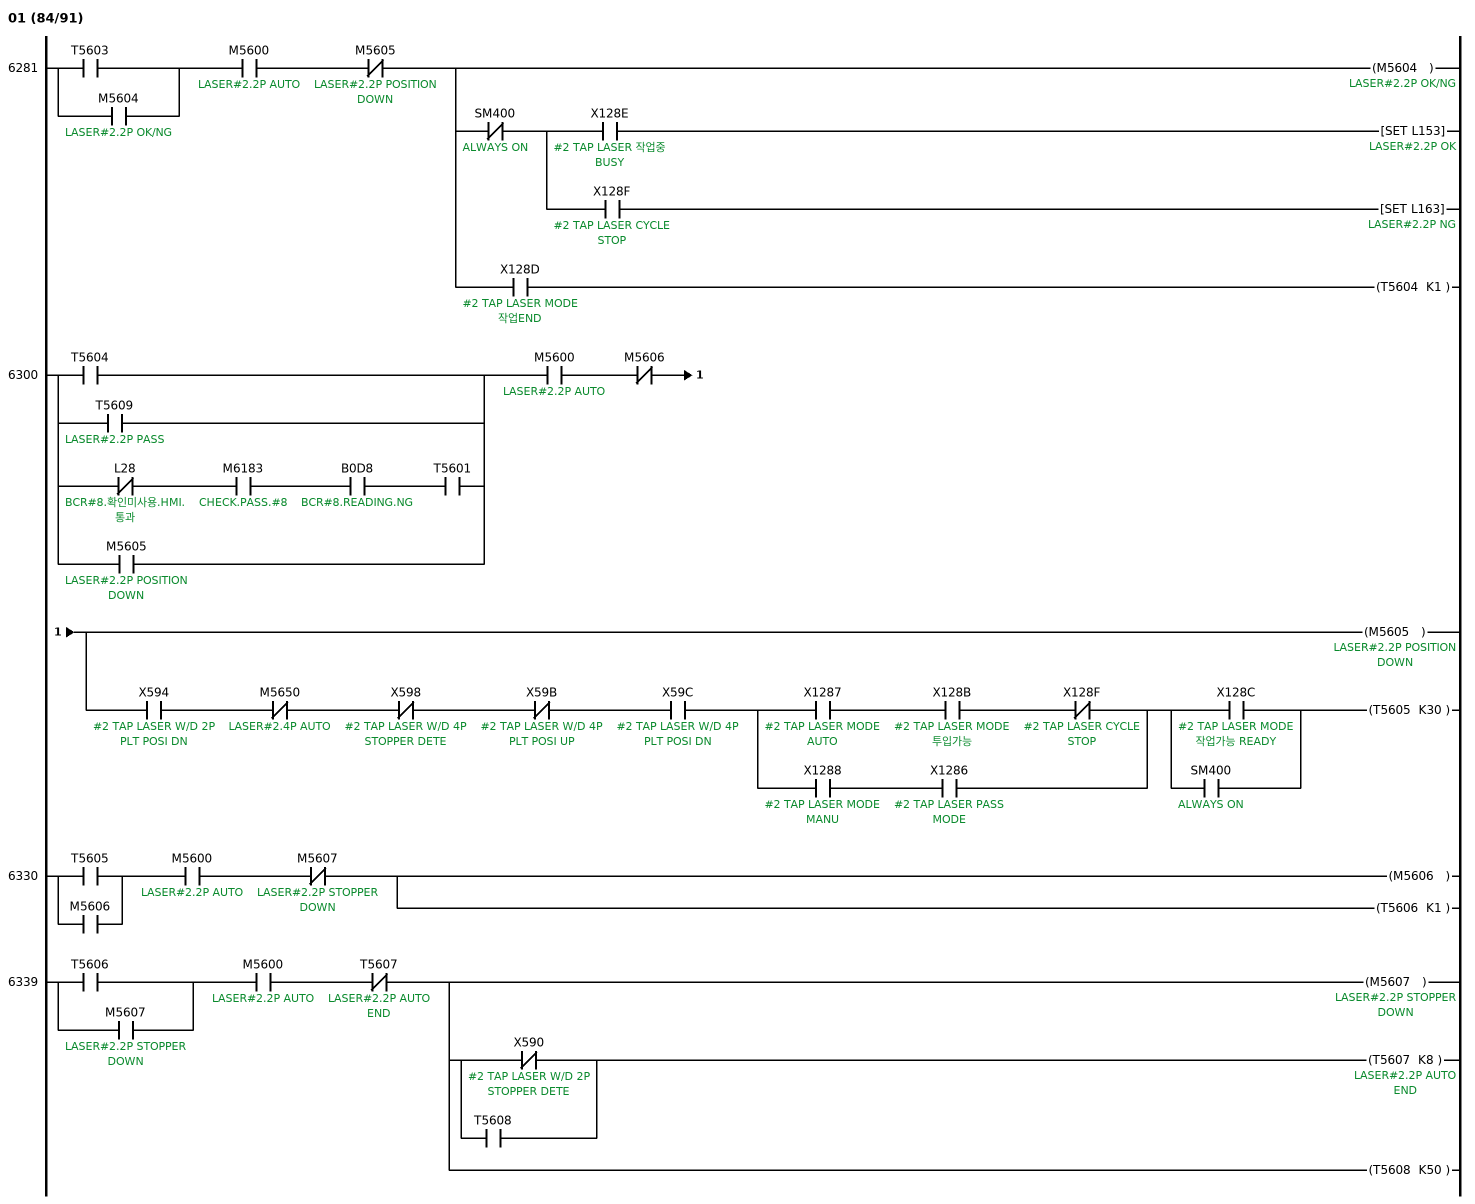
6281  LD      T5603
      OR      M5604  ; LASER#2.2P OK/NG
      AND     M5600  ; LASER#2.2P AUTO
      ANI     M5605  ; LASER#2.2P POSITION DOWN
      OUT     M5604  ; LASER#2.2P OK/NG
      MPS
      ANI     SM400  ; ALWAYS ON
      MPS
      AND     X128E  ; #2 TAP LASER 작업중 BUSY
      SET     L153  ; LASER#2.2P OK
      MPP
      AND     X128F  ; #2 TAP LASER CYCLE STOP
      SET     L163  ; LASER#2.2P NG
      MPP
      AND     X128D  ; #2 TAP LASER MODE 작업END
      OUT     T5604 K1
6300  LD      T5604
      OR      T5609  ; LASER#2.2P PASS
      LDI     L28  ; BCR#8.확인미사용.HMI.통과
      AND     M6183  ; CHECK.PASS.#8
      AND     B0D8  ; BCR#8.READING.NG
      AND     T5601
      ORB
      OR      M5605  ; LASER#2.2P POSITION DOWN
      AND     M5600  ; LASER#2.2P AUTO
      ANI     M5606
      OUT     M5605  ; LASER#2.2P POSITION DOWN
      AND     X594  ; #2 TAP LASER W/D 2P PLT POSI DN
      ANI     M5650  ; LASER#2.4P AUTO
      ANI     X598  ; #2 TAP LASER W/D 4P STOPPER DETE
      ANI     X59B  ; #2 TAP LASER W/D 4P PLT POSI UP
      AND     X59C  ; #2 TAP LASER W/D 4P PLT POSI DN
      LD      X1287  ; #2 TAP LASER MODE AUTO
      AND     X128B  ; #2 TAP LASER MODE 투입가능
      ANI     X128F  ; #2 TAP LASER CYCLE STOP
      LD      X1288  ; #2 TAP LASER MODE MANU
      AND     X1286  ; #2 TAP LASER PASS MODE
      ORB
      ANB
      LD      X128C  ; #2 TAP LASER MODE 작업가능 READY
      OR      SM400  ; ALWAYS ON
      ANB
      OUT     T5605 K30
6330  LD      T5605
      OR      M5606
      AND     M5600  ; LASER#2.2P AUTO
      ANI     M5607  ; LASER#2.2P STOPPER DOWN
      OUT     M5606
      OUT     T5606 K1
6339  LD      T5606
      OR      M5607  ; LASER#2.2P STOPPER DOWN
      AND     M5600  ; LASER#2.2P AUTO
      ANI     T5607  ; LASER#2.2P AUTO END
      OUT     M5607  ; LASER#2.2P STOPPER DOWN
      MPS
      LDI     X590  ; #2 TAP LASER W/D 2P STOPPER DETE
      OR      T5608
      ANB
      OUT     T5607 K8  ; LASER#2.2P AUTO END
      MPP
      OUT     T5608 K50
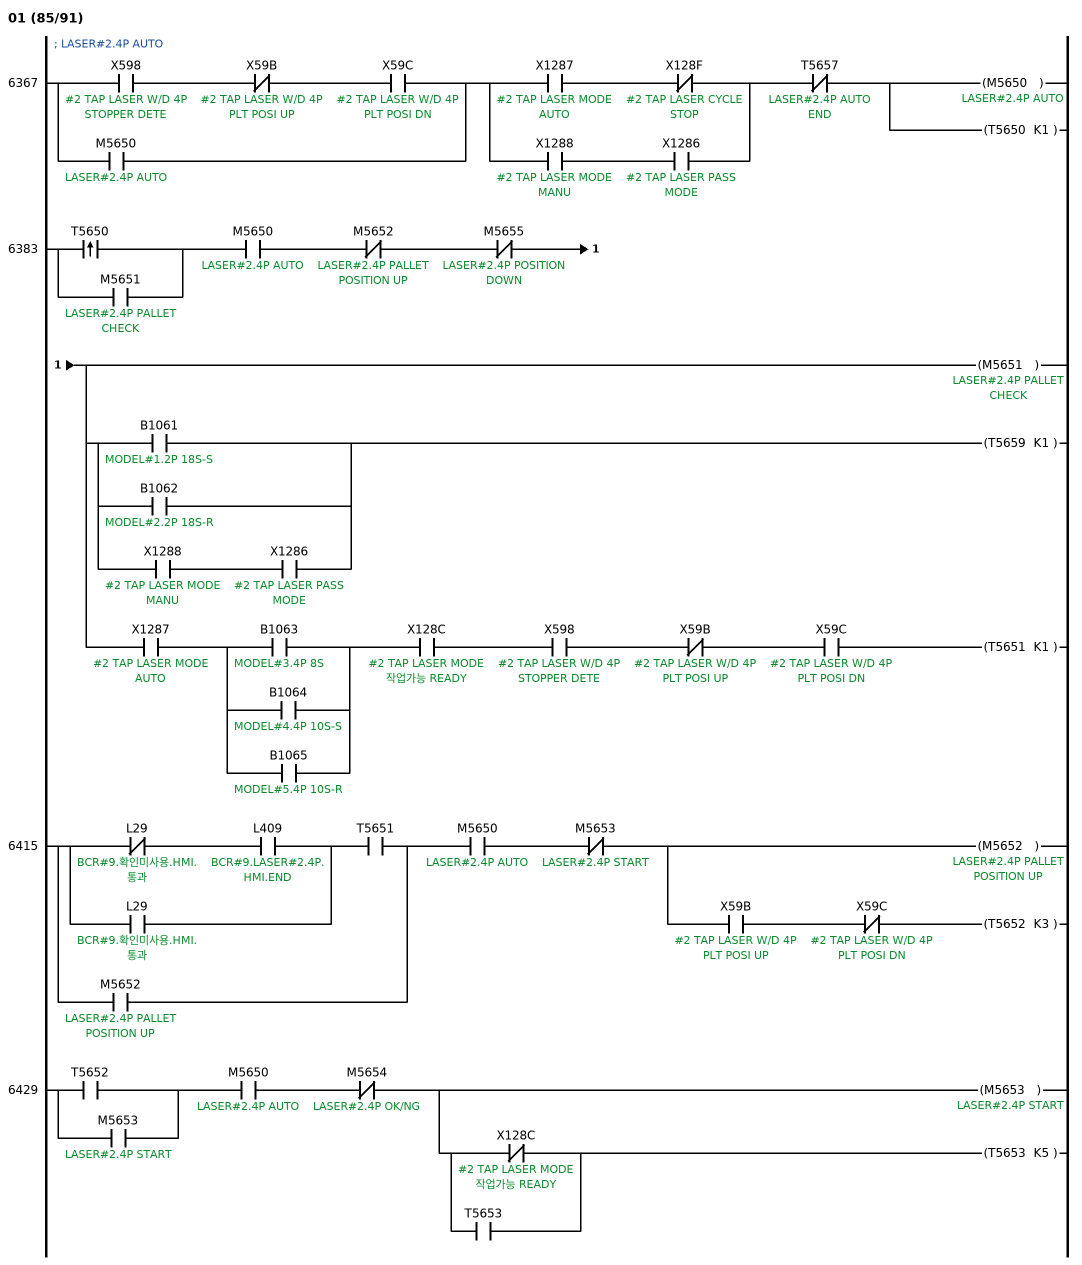
; LASER#2.4P AUTO
6367  LD      X598  ; #2 TAP LASER W/D 4P STOPPER DETE
      ANI     X59B  ; #2 TAP LASER W/D 4P PLT POSI UP
      AND     X59C  ; #2 TAP LASER W/D 4P PLT POSI DN
      OR      M5650  ; LASER#2.4P AUTO
      LD      X1287  ; #2 TAP LASER MODE AUTO
      ANI     X128F  ; #2 TAP LASER CYCLE STOP
      LD      X1288  ; #2 TAP LASER MODE MANU
      AND     X1286  ; #2 TAP LASER PASS MODE
      ORB
      ANB
      ANI     T5657  ; LASER#2.4P AUTO END
      OUT     M5650  ; LASER#2.4P AUTO
      OUT     T5650 K1
6383  LDP     T5650
      OR      M5651  ; LASER#2.4P PALLET CHECK
      AND     M5650  ; LASER#2.4P AUTO
      ANI     M5652  ; LASER#2.4P PALLET POSITION UP
      ANI     M5655  ; LASER#2.4P POSITION DOWN
      OUT     M5651  ; LASER#2.4P PALLET CHECK
      MPS
      LD      B1061  ; MODEL#1.2P 18S-S
      OR      B1062  ; MODEL#2.2P 18S-R
      LD      X1288  ; #2 TAP LASER MODE MANU
      AND     X1286  ; #2 TAP LASER PASS MODE
      ORB
      ANB
      OUT     T5659 K1
      MPP
      AND     X1287  ; #2 TAP LASER MODE AUTO
      LD      B1063  ; MODEL#3.4P 8S
      OR      B1064  ; MODEL#4.4P 10S-S
      OR      B1065  ; MODEL#5.4P 10S-R
      ANB
      AND     X128C  ; #2 TAP LASER MODE 작업가능 READY
      AND     X598  ; #2 TAP LASER W/D 4P STOPPER DETE
      ANI     X59B  ; #2 TAP LASER W/D 4P PLT POSI UP
      AND     X59C  ; #2 TAP LASER W/D 4P PLT POSI DN
      OUT     T5651 K1
6415  LDI     L29  ; BCR#9.확인미사용.HMI.통과
      AND     L409  ; BCR#9.LASER#2.4P.HMI.END
      OR      L29  ; BCR#9.확인미사용.HMI.통과
      AND     T5651
      OR      M5652  ; LASER#2.4P PALLET POSITION UP
      AND     M5650  ; LASER#2.4P AUTO
      ANI     M5653  ; LASER#2.4P START
      OUT     M5652  ; LASER#2.4P PALLET POSITION UP
      AND     X59B  ; #2 TAP LASER W/D 4P PLT POSI UP
      ANI     X59C  ; #2 TAP LASER W/D 4P PLT POSI DN
      OUT     T5652 K3
6429  LD      T5652
      OR      M5653  ; LASER#2.4P START
      AND     M5650  ; LASER#2.4P AUTO
      ANI     M5654  ; LASER#2.4P OK/NG
      OUT     M5653  ; LASER#2.4P START
      LDI     X128C  ; #2 TAP LASER MODE 작업가능 READY
      OR      T5653
      ANB
      OUT     T5653 K5
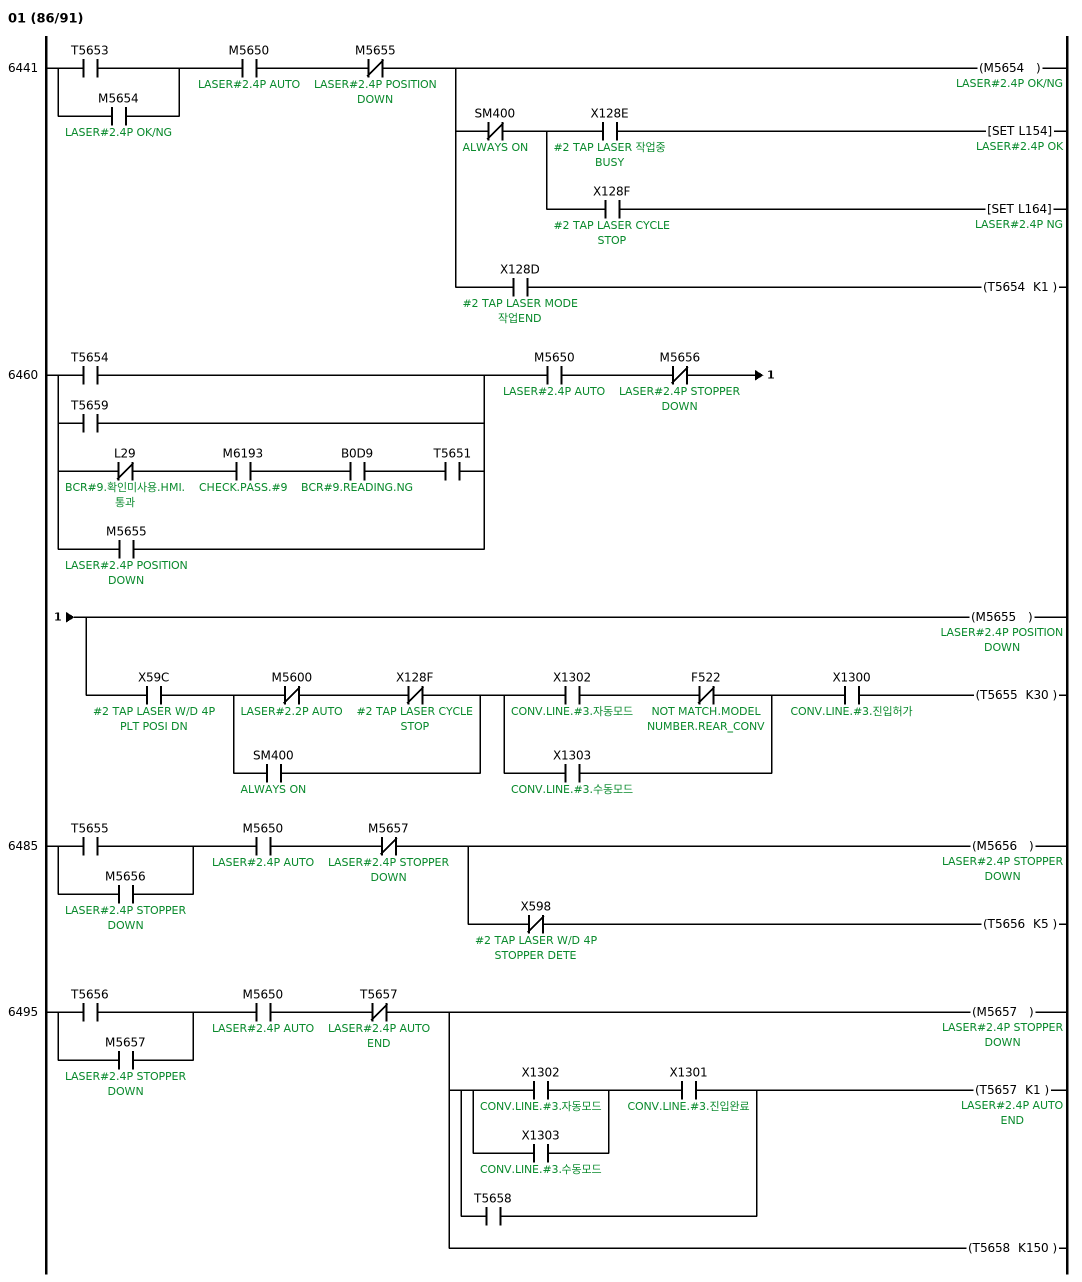
6441  LD      T5653
      OR      M5654  ; LASER#2.4P OK/NG
      AND     M5650  ; LASER#2.4P AUTO
      ANI     M5655  ; LASER#2.4P POSITION DOWN
      OUT     M5654  ; LASER#2.4P OK/NG
      MPS
      ANI     SM400  ; ALWAYS ON
      MPS
      AND     X128E  ; #2 TAP LASER 작업중 BUSY
      SET     L154  ; LASER#2.4P OK
      MPP
      AND     X128F  ; #2 TAP LASER CYCLE STOP
      SET     L164  ; LASER#2.4P NG
      MPP
      AND     X128D  ; #2 TAP LASER MODE 작업END
      OUT     T5654 K1
6460  LD      T5654
      OR      T5659
      LDI     L29  ; BCR#9.확인미사용.HMI.통과
      AND     M6193  ; CHECK.PASS.#9
      AND     B0D9  ; BCR#9.READING.NG
      AND     T5651
      ORB
      OR      M5655  ; LASER#2.4P POSITION DOWN
      AND     M5650  ; LASER#2.4P AUTO
      ANI     M5656  ; LASER#2.4P STOPPER DOWN
      OUT     M5655  ; LASER#2.4P POSITION DOWN
      AND     X59C  ; #2 TAP LASER W/D 4P PLT POSI DN
      LDI     M5600  ; LASER#2.2P AUTO
      ANI     X128F  ; #2 TAP LASER CYCLE STOP
      OR      SM400  ; ALWAYS ON
      ANB
      LD      X1302  ; CONV.LINE.#3.자동모드
      ANI     F522  ; NOT MATCH.MODEL NUMBER.REAR_CONV
      OR      X1303  ; CONV.LINE.#3.수동모드
      ANB
      AND     X1300  ; CONV.LINE.#3.진입허가
      OUT     T5655 K30
6485  LD      T5655
      OR      M5656  ; LASER#2.4P STOPPER DOWN
      AND     M5650  ; LASER#2.4P AUTO
      ANI     M5657  ; LASER#2.4P STOPPER DOWN
      OUT     M5656  ; LASER#2.4P STOPPER DOWN
      ANI     X598  ; #2 TAP LASER W/D 4P STOPPER DETE
      OUT     T5656 K5
6495  LD      T5656
      OR      M5657  ; LASER#2.4P STOPPER DOWN
      AND     M5650  ; LASER#2.4P AUTO
      ANI     T5657  ; LASER#2.4P AUTO END
      OUT     M5657  ; LASER#2.4P STOPPER DOWN
      MPS
      LD      X1302  ; CONV.LINE.#3.자동모드
      OR      X1303  ; CONV.LINE.#3.수동모드
      AND     X1301  ; CONV.LINE.#3.진입완료
      OR      T5658
      ANB
      OUT     T5657 K1  ; LASER#2.4P AUTO END
      MPP
      OUT     T5658 K150
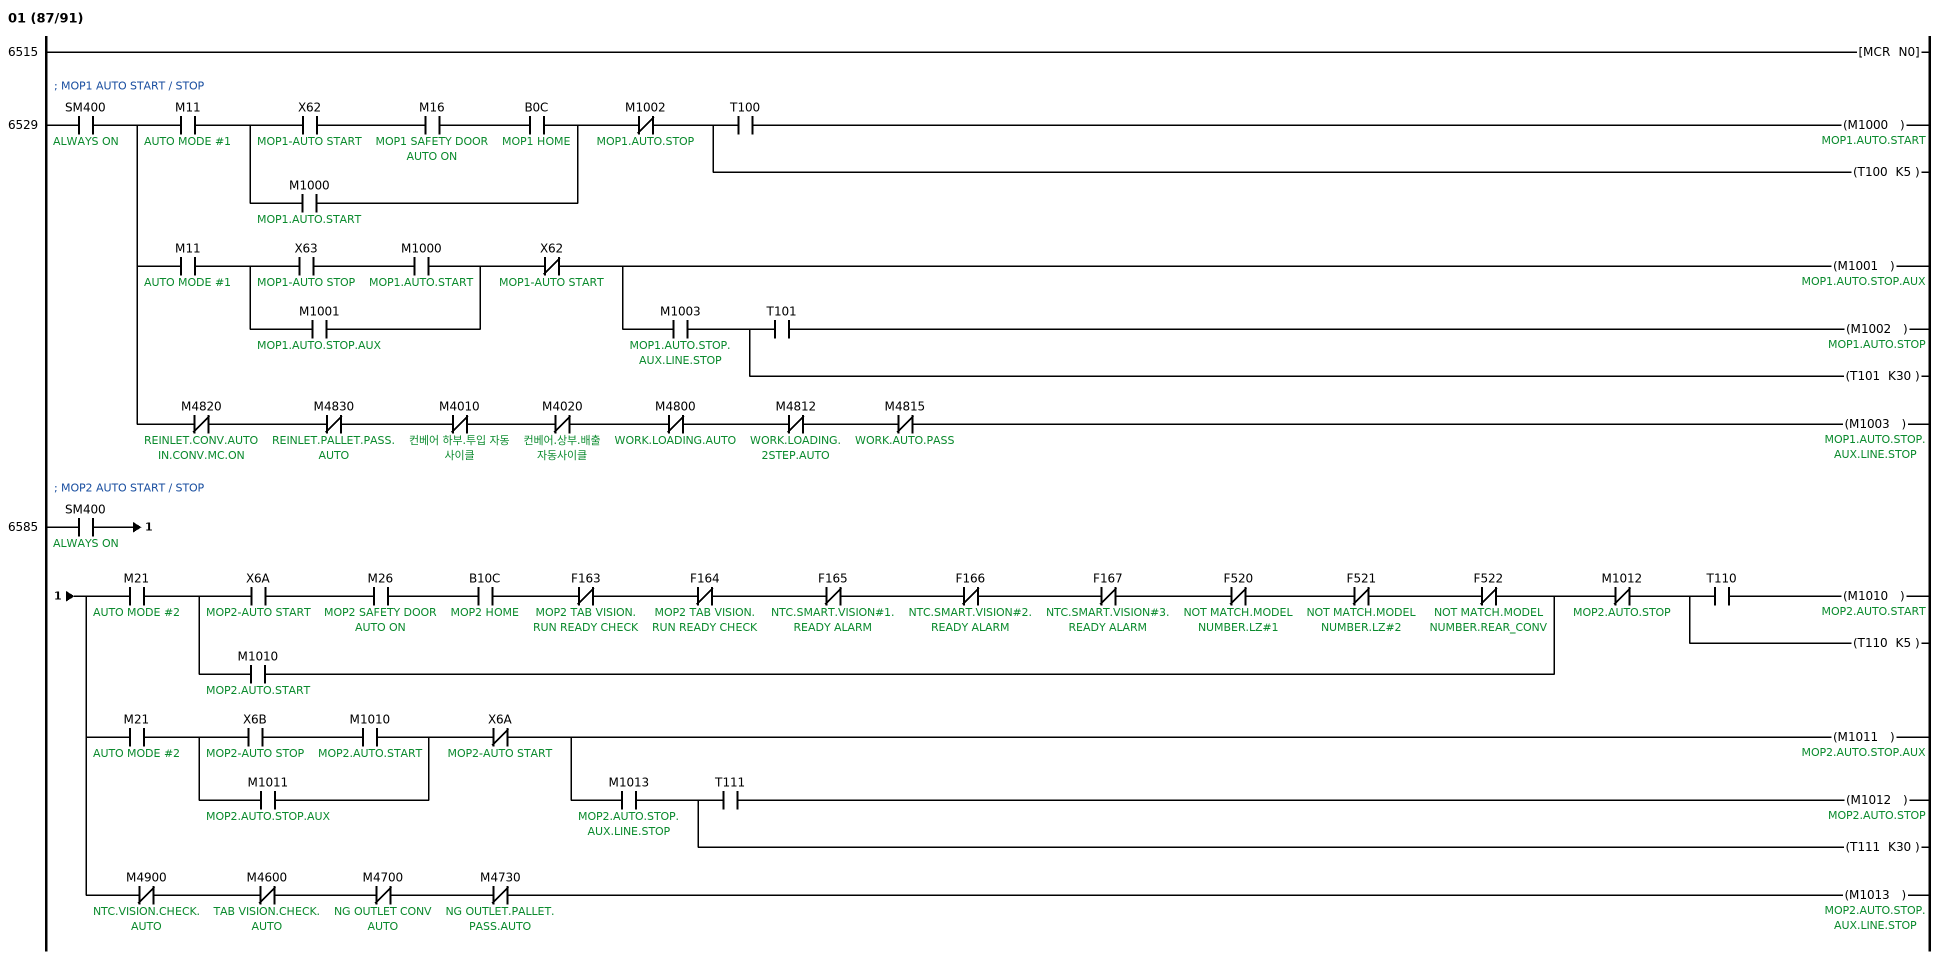
6515  MCR     N0
; MOP1 AUTO START / STOP
6529  LD      SM400  ; ALWAYS ON
      MPS
      AND     M11  ; AUTO MODE #1
      LD      X62  ; MOP1-AUTO START
      AND     M16  ; MOP1 SAFETY DOOR AUTO ON
      AND     B0C  ; MOP1 HOME
      OR      M1000  ; MOP1.AUTO.START
      ANB
      ANI     M1002  ; MOP1.AUTO.STOP
      MPS
      AND     T100
      OUT     M1000  ; MOP1.AUTO.START
      MPP
      OUT     T100 K5
      MRD
      AND     M11  ; AUTO MODE #1
      LD      X63  ; MOP1-AUTO STOP
      AND     M1000  ; MOP1.AUTO.START
      OR      M1001  ; MOP1.AUTO.STOP.AUX
      ANB
      ANI     X62  ; MOP1-AUTO START
      OUT     M1001  ; MOP1.AUTO.STOP.AUX
      AND     M1003  ; MOP1.AUTO.STOP.AUX.LINE.STOP
      MPS
      AND     T101
      OUT     M1002  ; MOP1.AUTO.STOP
      MPP
      OUT     T101 K30
      MPP
      ANI     M4820  ; REINLET.CONV.AUTO IN.CONV.MC.ON
      ANI     M4830  ; REINLET.PALLET.PASS.AUTO
      ANI     M4010  ; 컨베어 하부.투입 자동 사이클
      ANI     M4020  ; 컨베어.상부.배출 자동사이클
      ANI     M4800  ; WORK.LOADING.AUTO
      ANI     M4812  ; WORK.LOADING.2STEP.AUTO
      ANI     M4815  ; WORK.AUTO.PASS
      OUT     M1003  ; MOP1.AUTO.STOP.AUX.LINE.STOP
; MOP2 AUTO START / STOP
6585  LD      SM400  ; ALWAYS ON
      MPS
      AND     M21  ; AUTO MODE #2
      LD      X6A  ; MOP2-AUTO START
      AND     M26  ; MOP2 SAFETY DOOR AUTO ON
      AND     B10C  ; MOP2 HOME
      ANI     F163  ; MOP2 TAB VISION. RUN READY CHECK
      ANI     F164  ; MOP2 TAB VISION. RUN READY CHECK
      ANI     F165  ; NTC.SMART.VISION#1.READY ALARM
      ANI     F166  ; NTC.SMART.VISION#2.READY ALARM
      ANI     F167  ; NTC.SMART.VISION#3.READY ALARM
      ANI     F520  ; NOT MATCH.MODEL NUMBER.LZ#1
      ANI     F521  ; NOT MATCH.MODEL NUMBER.LZ#2
      ANI     F522  ; NOT MATCH.MODEL NUMBER.REAR_CONV
      OR      M1010  ; MOP2.AUTO.START
      ANB
      ANI     M1012  ; MOP2.AUTO.STOP
      MPS
      AND     T110
      OUT     M1010  ; MOP2.AUTO.START
      MPP
      OUT     T110 K5
      MRD
      AND     M21  ; AUTO MODE #2
      LD      X6B  ; MOP2-AUTO STOP
      AND     M1010  ; MOP2.AUTO.START
      OR      M1011  ; MOP2.AUTO.STOP.AUX
      ANB
      ANI     X6A  ; MOP2-AUTO START
      OUT     M1011  ; MOP2.AUTO.STOP.AUX
      AND     M1013  ; MOP2.AUTO.STOP.AUX.LINE.STOP
      MPS
      AND     T111
      OUT     M1012  ; MOP2.AUTO.STOP
      MPP
      OUT     T111 K30
      MPP
      ANI     M4900  ; NTC.VISION.CHECK.AUTO
      ANI     M4600  ; TAB VISION.CHECK.AUTO
      ANI     M4700  ; NG OUTLET CONV AUTO
      ANI     M4730  ; NG OUTLET.PALLET.PASS.AUTO
      OUT     M1013  ; MOP2.AUTO.STOP.AUX.LINE.STOP
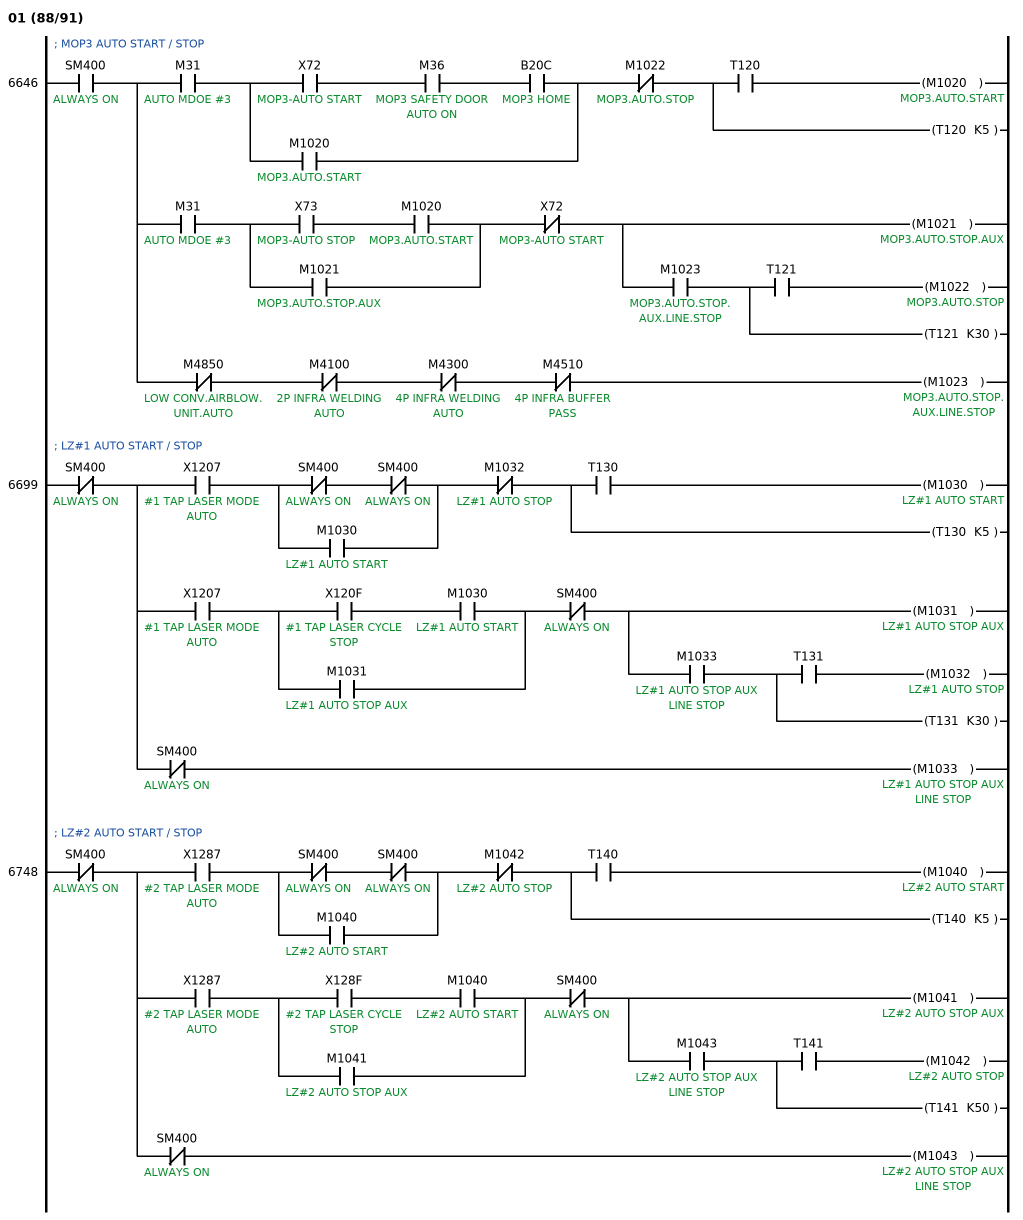
; MOP3 AUTO START / STOP
6646  LD      SM400  ; ALWAYS ON
      MPS
      AND     M31  ; AUTO MDOE #3
      LD      X72  ; MOP3-AUTO START
      AND     M36  ; MOP3 SAFETY DOOR AUTO ON
      AND     B20C  ; MOP3 HOME
      OR      M1020  ; MOP3.AUTO.START
      ANB
      ANI     M1022  ; MOP3.AUTO.STOP
      MPS
      AND     T120
      OUT     M1020  ; MOP3.AUTO.START
      MPP
      OUT     T120 K5
      MRD
      AND     M31  ; AUTO MDOE #3
      LD      X73  ; MOP3-AUTO STOP
      AND     M1020  ; MOP3.AUTO.START
      OR      M1021  ; MOP3.AUTO.STOP.AUX
      ANB
      ANI     X72  ; MOP3-AUTO START
      OUT     M1021  ; MOP3.AUTO.STOP.AUX
      AND     M1023  ; MOP3.AUTO.STOP.AUX.LINE.STOP
      MPS
      AND     T121
      OUT     M1022  ; MOP3.AUTO.STOP
      MPP
      OUT     T121 K30
      MPP
      ANI     M4850  ; LOW CONV.AIRBLOW.UNIT.AUTO
      ANI     M4100  ; 2P INFRA WELDING AUTO
      ANI     M4300  ; 4P INFRA WELDING AUTO
      ANI     M4510  ; 4P INFRA BUFFER PASS
      OUT     M1023  ; MOP3.AUTO.STOP.AUX.LINE.STOP
; LZ#1 AUTO START / STOP
6699  LDI     SM400  ; ALWAYS ON
      MPS
      AND     X1207  ; #1 TAP LASER MODE AUTO
      LDI     SM400  ; ALWAYS ON
      ANI     SM400  ; ALWAYS ON
      OR      M1030  ; LZ#1 AUTO START
      ANB
      ANI     M1032  ; LZ#1 AUTO STOP
      MPS
      AND     T130
      OUT     M1030  ; LZ#1 AUTO START
      MPP
      OUT     T130 K5
      MRD
      AND     X1207  ; #1 TAP LASER MODE AUTO
      LD      X120F  ; #1 TAP LASER CYCLE STOP
      AND     M1030  ; LZ#1 AUTO START
      OR      M1031  ; LZ#1 AUTO STOP AUX
      ANB
      ANI     SM400  ; ALWAYS ON
      OUT     M1031  ; LZ#1 AUTO STOP AUX
      AND     M1033  ; LZ#1 AUTO STOP AUX LINE STOP
      MPS
      AND     T131
      OUT     M1032  ; LZ#1 AUTO STOP
      MPP
      OUT     T131 K30
      MPP
      ANI     SM400  ; ALWAYS ON
      OUT     M1033  ; LZ#1 AUTO STOP AUX LINE STOP
; LZ#2 AUTO START / STOP
6748  LDI     SM400  ; ALWAYS ON
      MPS
      AND     X1287  ; #2 TAP LASER MODE AUTO
      LDI     SM400  ; ALWAYS ON
      ANI     SM400  ; ALWAYS ON
      OR      M1040  ; LZ#2 AUTO START
      ANB
      ANI     M1042  ; LZ#2 AUTO STOP
      MPS
      AND     T140
      OUT     M1040  ; LZ#2 AUTO START
      MPP
      OUT     T140 K5
      MRD
      AND     X1287  ; #2 TAP LASER MODE AUTO
      LD      X128F  ; #2 TAP LASER CYCLE STOP
      AND     M1040  ; LZ#2 AUTO START
      OR      M1041  ; LZ#2 AUTO STOP AUX
      ANB
      ANI     SM400  ; ALWAYS ON
      OUT     M1041  ; LZ#2 AUTO STOP AUX
      AND     M1043  ; LZ#2 AUTO STOP AUX LINE STOP
      MPS
      AND     T141
      OUT     M1042  ; LZ#2 AUTO STOP
      MPP
      OUT     T141 K50
      MPP
      ANI     SM400  ; ALWAYS ON
      OUT     M1043  ; LZ#2 AUTO STOP AUX LINE STOP
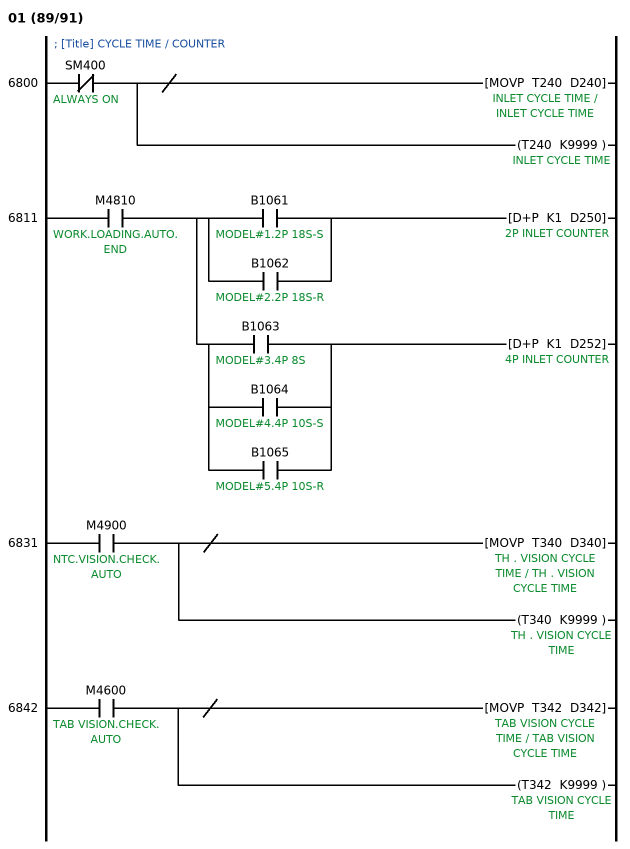
; [Title] CYCLE TIME / COUNTER
6800  LDI     SM400  ; ALWAYS ON
      MPS
      INV
      MOVP    T240 D240  ; INLET CYCLE TIME / INLET CYCLE TIME
      MPP
      OUT     T240 K9999  ; INLET CYCLE TIME
6811  LD      M4810  ; WORK.LOADING.AUTO.END
      MPS
      LD      B1061  ; MODEL#1.2P 18S-S
      OR      B1062  ; MODEL#2.2P 18S-R
      ANB
      D+P     K1 D250  ; 2P INLET COUNTER
      MPP
      LD      B1063  ; MODEL#3.4P 8S
      OR      B1064  ; MODEL#4.4P 10S-S
      OR      B1065  ; MODEL#5.4P 10S-R
      ANB
      D+P     K1 D252  ; 4P INLET COUNTER
6831  LD      M4900  ; NTC.VISION.CHECK.AUTO
      MPS
      INV
      MOVP    T340 D340  ; TH . VISION CYCLE TIME / TH . VISION CYCLE TIME
      MPP
      OUT     T340 K9999  ; TH . VISION CYCLE TIME
6842  LD      M4600  ; TAB VISION.CHECK.AUTO
      MPS
      INV
      MOVP    T342 D342  ; TAB VISION CYCLE TIME / TAB VISION CYCLE TIME
      MPP
      OUT     T342 K9999  ; TAB VISION CYCLE TIME
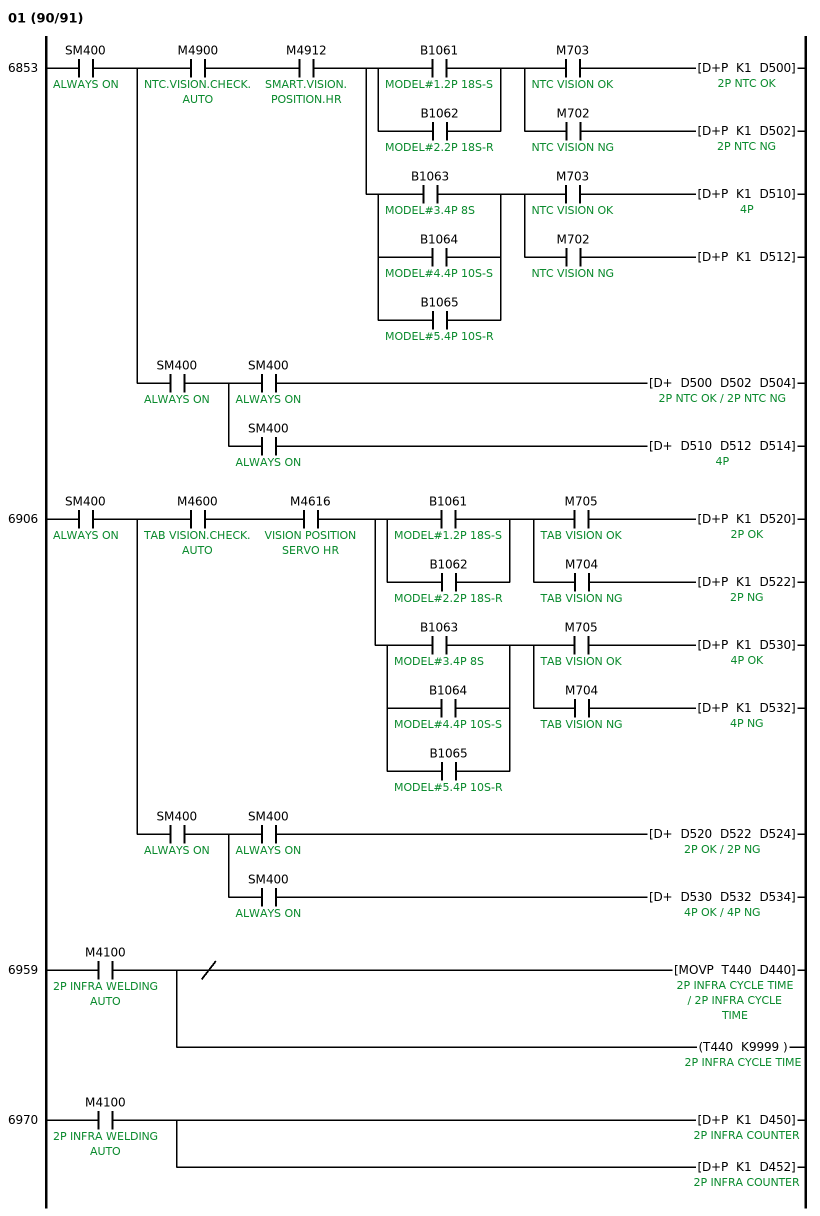
6853  LD      SM400  ; ALWAYS ON
      MPS
      AND     M4900  ; NTC.VISION.CHECK.AUTO
      AND     M4912  ; SMART.VISION.POSITION.HR
      MPS
      LD      B1061  ; MODEL#1.2P 18S-S
      OR      B1062  ; MODEL#2.2P 18S-R
      ANB
      MPS
      AND     M703  ; NTC VISION OK
      D+P     K1 D500  ; 2P NTC OK
      MPP
      AND     M702  ; NTC VISION NG
      D+P     K1 D502  ; 2P NTC NG
      MPP
      LD      B1063  ; MODEL#3.4P 8S
      OR      B1064  ; MODEL#4.4P 10S-S
      OR      B1065  ; MODEL#5.4P 10S-R
      ANB
      MPS
      AND     M703  ; NTC VISION OK
      D+P     K1 D510  ; 4P
      MPP
      AND     M702  ; NTC VISION NG
      D+P     K1 D512
      MPP
      AND     SM400  ; ALWAYS ON
      MPS
      AND     SM400  ; ALWAYS ON
      D+      D500 D502 D504
      MPP
      AND     SM400  ; ALWAYS ON
      D+      D510 D512 D514
6906  LD      SM400  ; ALWAYS ON
      MPS
      AND     M4600  ; TAB VISION.CHECK.AUTO
      AND     M4616  ; VISION POSITION SERVO HR
      MPS
      LD      B1061  ; MODEL#1.2P 18S-S
      OR      B1062  ; MODEL#2.2P 18S-R
      ANB
      MPS
      AND     M705  ; TAB VISION OK
      D+P     K1 D520  ; 2P OK
      MPP
      AND     M704  ; TAB VISION NG
      D+P     K1 D522  ; 2P NG
      MPP
      LD      B1063  ; MODEL#3.4P 8S
      OR      B1064  ; MODEL#4.4P 10S-S
      OR      B1065  ; MODEL#5.4P 10S-R
      ANB
      MPS
      AND     M705  ; TAB VISION OK
      D+P     K1 D530  ; 4P OK
      MPP
      AND     M704  ; TAB VISION NG
      D+P     K1 D532  ; 4P NG
      MPP
      AND     SM400  ; ALWAYS ON
      MPS
      AND     SM400  ; ALWAYS ON
      D+      D520 D522 D524
      MPP
      AND     SM400  ; ALWAYS ON
      D+      D530 D532 D534
6959  LD      M4100  ; 2P INFRA WELDING AUTO
      MPS
      INV
      MOVP    T440 D440  ; 2P INFRA CYCLE TIME / 2P INFRA CYCLE TIME
      MPP
      OUT     T440 K9999  ; 2P INFRA CYCLE TIME
6970  LD      M4100  ; 2P INFRA WELDING AUTO
      D+P     K1 D450  ; 2P INFRA COUNTER
      D+P     K1 D452  ; 2P INFRA COUNTER
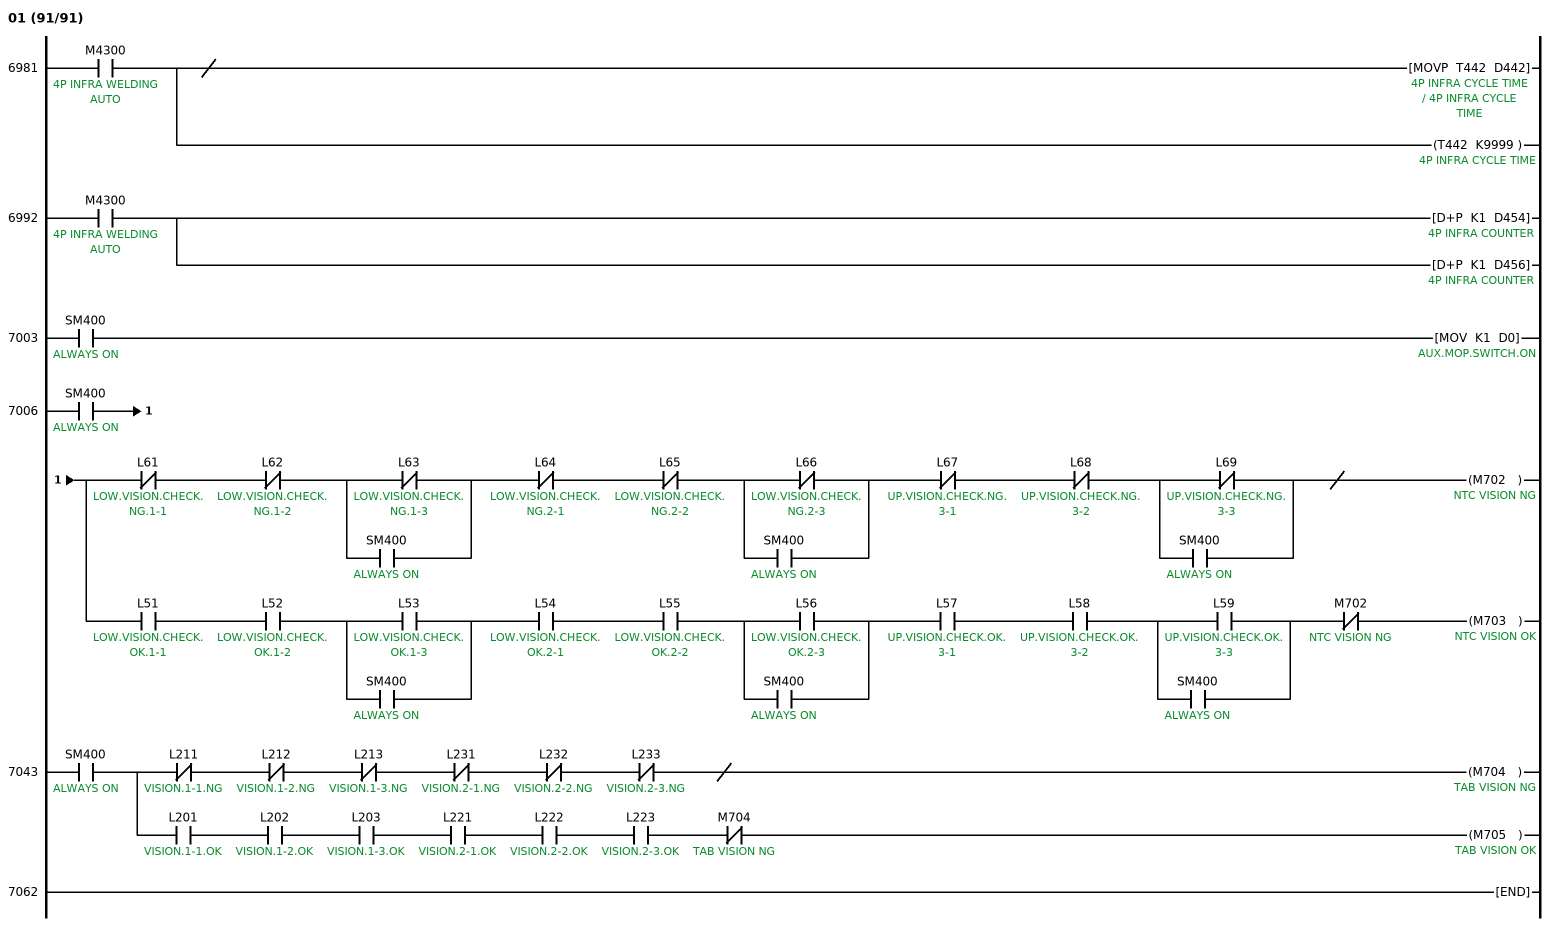
6981  LD      M4300  ; 4P INFRA WELDING AUTO
      MPS
      INV
      MOVP    T442 D442  ; 4P INFRA CYCLE TIME / 4P INFRA CYCLE TIME
      MPP
      OUT     T442 K9999  ; 4P INFRA CYCLE TIME
6992  LD      M4300  ; 4P INFRA WELDING AUTO
      D+P     K1 D454  ; 4P INFRA COUNTER
      D+P     K1 D456  ; 4P INFRA COUNTER
7003  LD      SM400  ; ALWAYS ON
      MOV     K1 D0  ; AUX.MOP.SWITCH.ON
7006  LD      SM400  ; ALWAYS ON
      MPS
      ANI     L61  ; LOW.VISION.CHECK.NG.1-1
      ANI     L62  ; LOW.VISION.CHECK.NG.1-2
      LDI     L63  ; LOW.VISION.CHECK.NG.1-3
      OR      SM400  ; ALWAYS ON
      ANB
      ANI     L64  ; LOW.VISION.CHECK.NG.2-1
      ANI     L65  ; LOW.VISION.CHECK.NG.2-2
      LDI     L66  ; LOW.VISION.CHECK.NG.2-3
      OR      SM400  ; ALWAYS ON
      ANB
      ANI     L67  ; UP.VISION.CHECK.NG.3-1
      ANI     L68  ; UP.VISION.CHECK.NG.3-2
      LDI     L69  ; UP.VISION.CHECK.NG.3-3
      OR      SM400  ; ALWAYS ON
      ANB
      INV
      OUT     M702  ; NTC VISION NG
      MPP
      AND     L51  ; LOW.VISION.CHECK.OK.1-1
      AND     L52  ; LOW.VISION.CHECK.OK.1-2
      LD      L53  ; LOW.VISION.CHECK.OK.1-3
      OR      SM400  ; ALWAYS ON
      ANB
      AND     L54  ; LOW.VISION.CHECK.OK.2-1
      AND     L55  ; LOW.VISION.CHECK.OK.2-2
      LD      L56  ; LOW.VISION.CHECK.OK.2-3
      OR      SM400  ; ALWAYS ON
      ANB
      AND     L57  ; UP.VISION.CHECK.OK.3-1
      AND     L58  ; UP.VISION.CHECK.OK.3-2
      LD      L59  ; UP.VISION.CHECK.OK.3-3
      OR      SM400  ; ALWAYS ON
      ANB
      ANI     M702  ; NTC VISION NG
      OUT     M703  ; NTC VISION OK
7043  LD      SM400  ; ALWAYS ON
      MPS
      ANI     L211  ; VISION.1-1.NG
      ANI     L212  ; VISION.1-2.NG
      ANI     L213  ; VISION.1-3.NG
      ANI     L231  ; VISION.2-1.NG
      ANI     L232  ; VISION.2-2.NG
      ANI     L233  ; VISION.2-3.NG
      INV
      OUT     M704  ; TAB VISION NG
      MPP
      AND     L201  ; VISION.1-1.OK
      AND     L202  ; VISION.1-2.OK
      AND     L203  ; VISION.1-3.OK
      AND     L221  ; VISION.2-1.OK
      AND     L222  ; VISION.2-2.OK
      AND     L223  ; VISION.2-3.OK
      ANI     M704  ; TAB VISION NG
      OUT     M705  ; TAB VISION OK
7062  END
END_PROGRAM

PROGRAM 05  // HMI
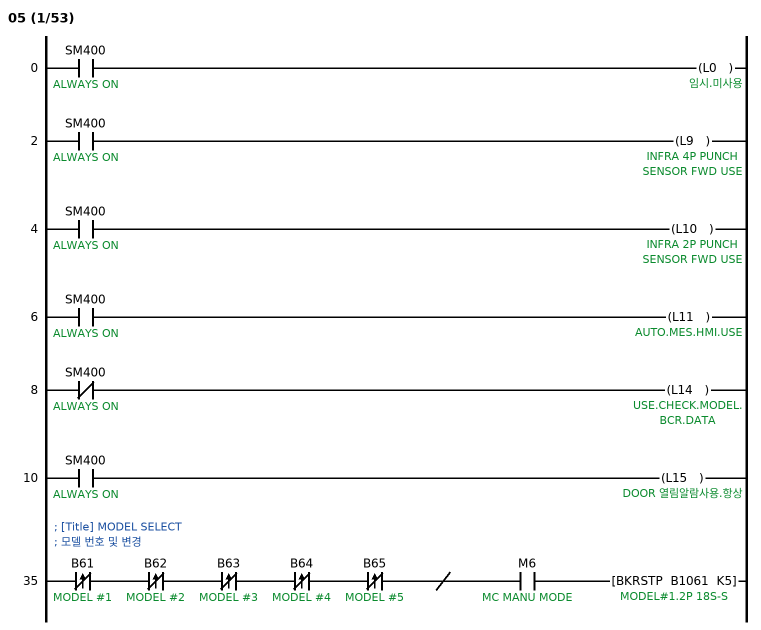
0     LD      SM400  ; ALWAYS ON
      OUT     L0  ; 임시.미사용
2     LD      SM400  ; ALWAYS ON
      OUT     L9  ; INFRA 4P PUNCH SENSOR FWD USE
4     LD      SM400  ; ALWAYS ON
      OUT     L10  ; INFRA 2P PUNCH SENSOR FWD USE
6     LD      SM400  ; ALWAYS ON
      OUT     L11  ; AUTO.MES.HMI.USE
8     LDI     SM400  ; ALWAYS ON
      OUT     L14  ; USE.CHECK.MODEL.BCR.DATA
10    LD      SM400  ; ALWAYS ON
      OUT     L15  ; DOOR 열림알람사용.항상
; [Title] MODEL SELECT
; 모델 번호 및 변경
35    LDPI    B61  ; MODEL #1
      ANDPI   B62  ; MODEL #2
      ANDPI   B63  ; MODEL #3
      ANDPI   B64  ; MODEL #4
      ANDPI   B65  ; MODEL #5
      INV
      AND     M6  ; MC MANU MODE
      BKRSTP  B1061 K5  ; MODEL#1.2P 18S-S
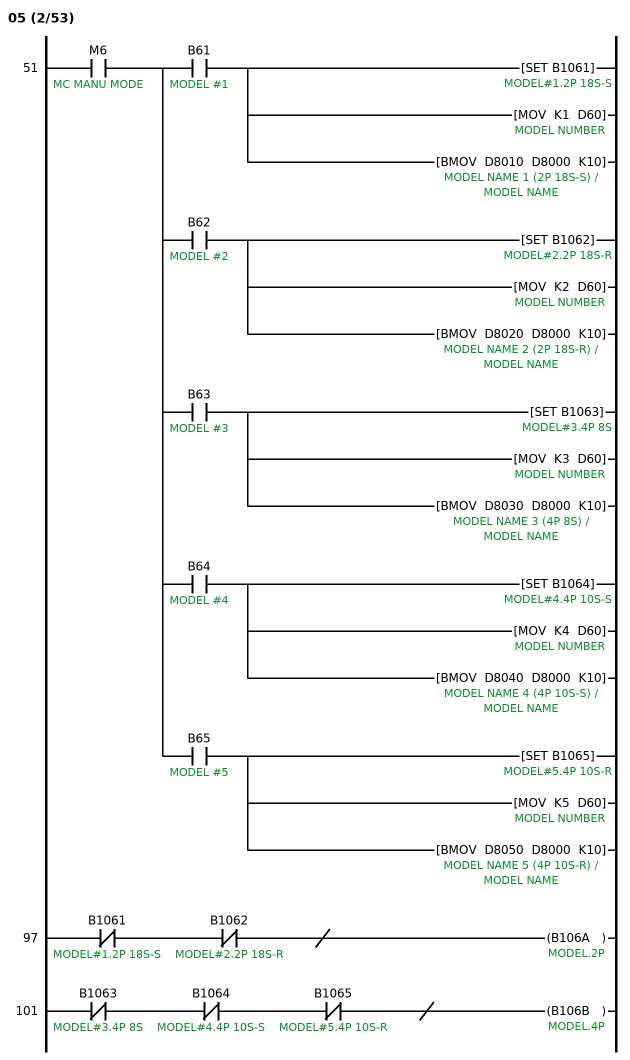
51    LD      M6  ; MC MANU MODE
      MPS
      AND     B61  ; MODEL #1
      SET     B1061  ; MODEL#1.2P 18S-S
      MOV     K1 D60  ; MODEL NUMBER
      BMOV    D8010 D8000 K10  ; MODEL NAME 1 (2P 18S-S) / MODEL NAME
      MRD
      AND     B62  ; MODEL #2
      SET     B1062  ; MODEL#2.2P 18S-R
      MOV     K2 D60
      BMOV    D8020 D8000 K10  ; MODEL NAME 2 (2P 18S-R)
      MRD
      AND     B63  ; MODEL #3
      SET     B1063  ; MODEL#3.4P 8S
      MOV     K3 D60
      BMOV    D8030 D8000 K10  ; MODEL NAME 3 (4P 8S)
      MRD
      AND     B64  ; MODEL #4
      SET     B1064  ; MODEL#4.4P 10S-S
      MOV     K4 D60
      BMOV    D8040 D8000 K10  ; MODEL NAME 4 (4P 10S-S)
      MPP
      AND     B65  ; MODEL #5
      SET     B1065  ; MODEL#5.4P 10S-R
      MOV     K5 D60
      BMOV    D8050 D8000 K10  ; MODEL NAME 5 (4P 10S-R)
97    LDI     B1061  ; MODEL#1.2P 18S-S
      ANI     B1062  ; MODEL#2.2P 18S-R
      INV
      OUT     B106A  ; MODEL.2P
101   LDI     B1063  ; MODEL#3.4P 8S
      ANI     B1064  ; MODEL#4.4P 10S-S
      ANI     B1065  ; MODEL#5.4P 10S-R
      INV
      OUT     B106B  ; MODEL.4P
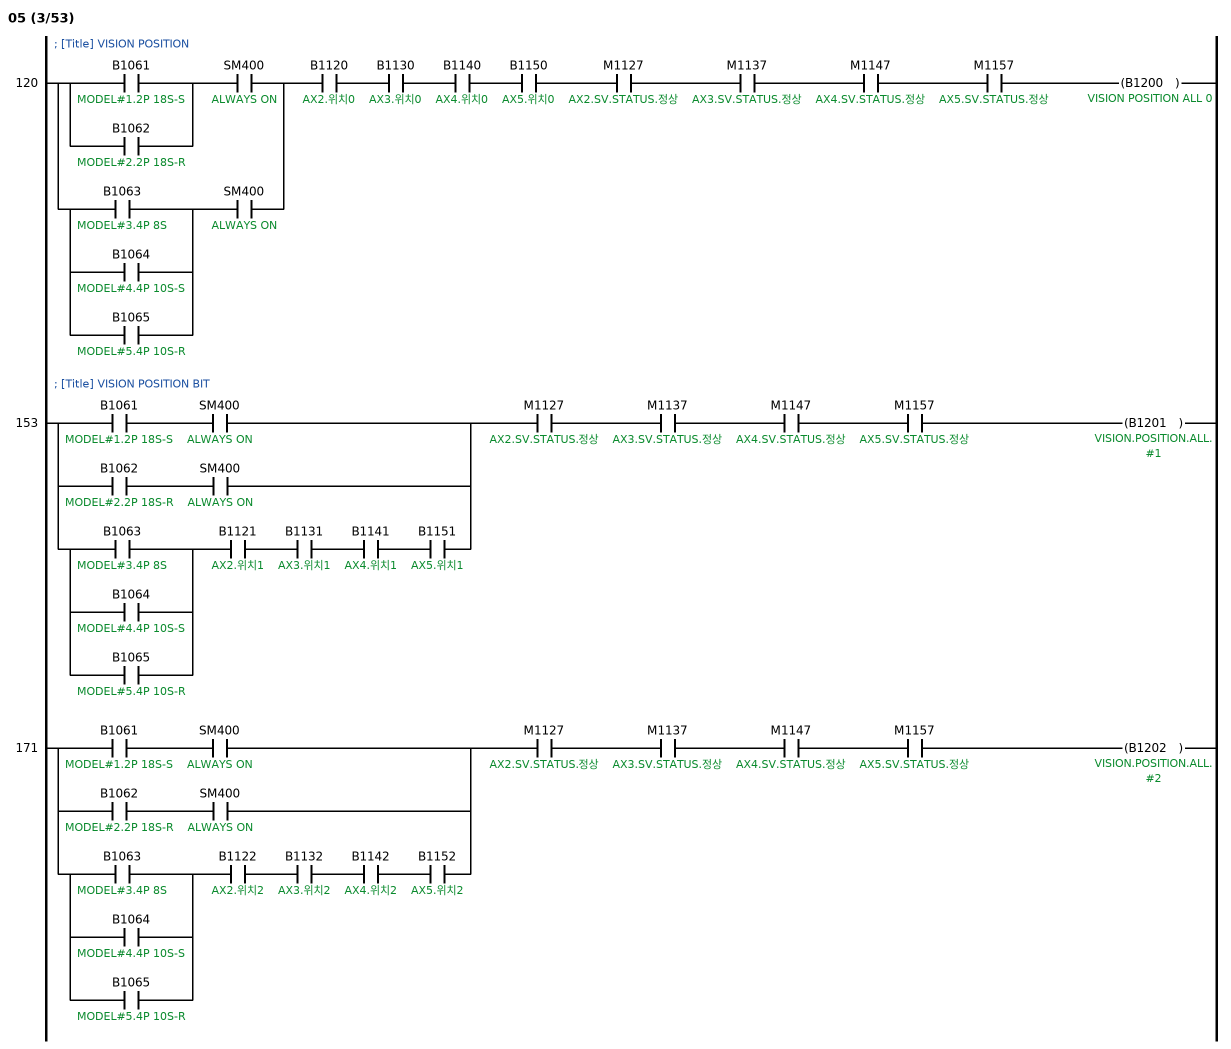
; [Title] VISION POSITION
120   LD      B1061  ; MODEL#1.2P 18S-S
      OR      B1062  ; MODEL#2.2P 18S-R
      AND     SM400  ; ALWAYS ON
      LD      B1063  ; MODEL#3.4P 8S
      OR      B1064  ; MODEL#4.4P 10S-S
      OR      B1065  ; MODEL#5.4P 10S-R
      AND     SM400  ; ALWAYS ON
      ORB
      AND     B1120  ; AX2.위치0
      AND     B1130  ; AX3.위치0
      AND     B1140  ; AX4.위치0
      AND     B1150  ; AX5.위치0
      AND     M1127  ; AX2.SV.STATUS.정상
      AND     M1137  ; AX3.SV.STATUS.정상
      AND     M1147  ; AX4.SV.STATUS.정상
      AND     M1157  ; AX5.SV.STATUS.정상
      OUT     B1200  ; VISION POSITION ALL 0
; [Title] VISION POSITION BIT
153   LD      B1061  ; MODEL#1.2P 18S-S
      AND     SM400  ; ALWAYS ON
      LD      B1062  ; MODEL#2.2P 18S-R
      AND     SM400  ; ALWAYS ON
      ORB
      LD      B1063  ; MODEL#3.4P 8S
      OR      B1064  ; MODEL#4.4P 10S-S
      OR      B1065  ; MODEL#5.4P 10S-R
      AND     B1121  ; AX2.위치1
      AND     B1131  ; AX3.위치1
      AND     B1141  ; AX4.위치1
      AND     B1151  ; AX5.위치1
      ORB
      AND     M1127  ; AX2.SV.STATUS.정상
      AND     M1137  ; AX3.SV.STATUS.정상
      AND     M1147  ; AX4.SV.STATUS.정상
      AND     M1157  ; AX5.SV.STATUS.정상
      OUT     B1201  ; VISION.POSITION.ALL.#1
171   LD      B1061  ; MODEL#1.2P 18S-S
      AND     SM400  ; ALWAYS ON
      LD      B1062  ; MODEL#2.2P 18S-R
      AND     SM400  ; ALWAYS ON
      ORB
      LD      B1063  ; MODEL#3.4P 8S
      OR      B1064  ; MODEL#4.4P 10S-S
      OR      B1065  ; MODEL#5.4P 10S-R
      AND     B1122  ; AX2.위치2
      AND     B1132  ; AX3.위치2
      AND     B1142  ; AX4.위치2
      AND     B1152  ; AX5.위치2
      ORB
      AND     M1127  ; AX2.SV.STATUS.정상
      AND     M1137  ; AX3.SV.STATUS.정상
      AND     M1147  ; AX4.SV.STATUS.정상
      AND     M1157  ; AX5.SV.STATUS.정상
      OUT     B1202  ; VISION.POSITION.ALL.#2
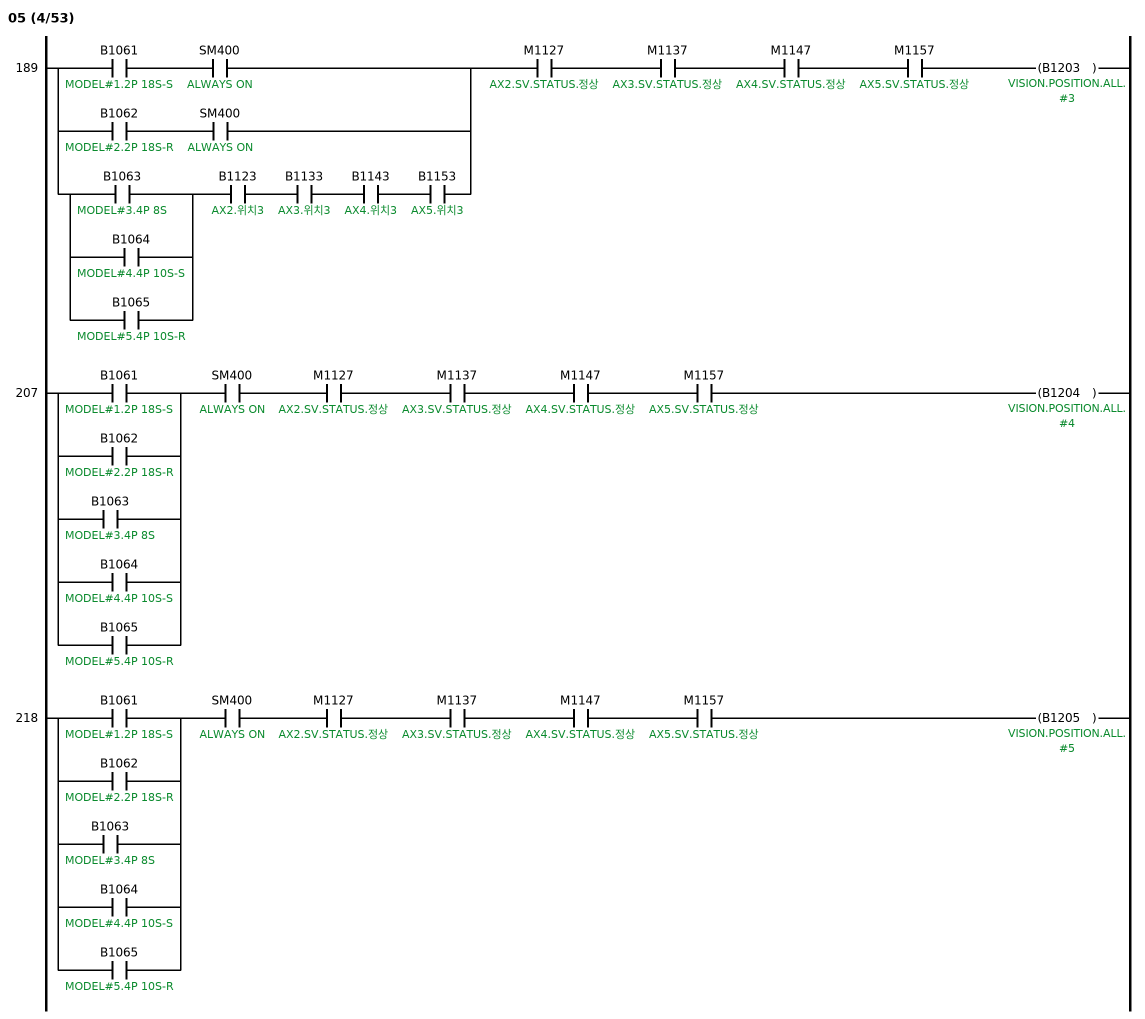
189   LD      B1061  ; MODEL#1.2P 18S-S
      AND     SM400  ; ALWAYS ON
      LD      B1062  ; MODEL#2.2P 18S-R
      AND     SM400  ; ALWAYS ON
      ORB
      LD      B1063  ; MODEL#3.4P 8S
      OR      B1064  ; MODEL#4.4P 10S-S
      OR      B1065  ; MODEL#5.4P 10S-R
      AND     B1123  ; AX2.위치3
      AND     B1133  ; AX3.위치3
      AND     B1143  ; AX4.위치3
      AND     B1153  ; AX5.위치3
      ORB
      AND     M1127  ; AX2.SV.STATUS.정상
      AND     M1137  ; AX3.SV.STATUS.정상
      AND     M1147  ; AX4.SV.STATUS.정상
      AND     M1157  ; AX5.SV.STATUS.정상
      OUT     B1203  ; VISION.POSITION.ALL.#3
207   LD      B1061  ; MODEL#1.2P 18S-S
      OR      B1062  ; MODEL#2.2P 18S-R
      OR      B1063  ; MODEL#3.4P 8S
      OR      B1064  ; MODEL#4.4P 10S-S
      OR      B1065  ; MODEL#5.4P 10S-R
      AND     SM400  ; ALWAYS ON
      AND     M1127  ; AX2.SV.STATUS.정상
      AND     M1137  ; AX3.SV.STATUS.정상
      AND     M1147  ; AX4.SV.STATUS.정상
      AND     M1157  ; AX5.SV.STATUS.정상
      OUT     B1204  ; VISION.POSITION.ALL.#4
218   LD      B1061  ; MODEL#1.2P 18S-S
      OR      B1062  ; MODEL#2.2P 18S-R
      OR      B1063  ; MODEL#3.4P 8S
      OR      B1064  ; MODEL#4.4P 10S-S
      OR      B1065  ; MODEL#5.4P 10S-R
      AND     SM400  ; ALWAYS ON
      AND     M1127  ; AX2.SV.STATUS.정상
      AND     M1137  ; AX3.SV.STATUS.정상
      AND     M1147  ; AX4.SV.STATUS.정상
      AND     M1157  ; AX5.SV.STATUS.정상
      OUT     B1205  ; VISION.POSITION.ALL.#5
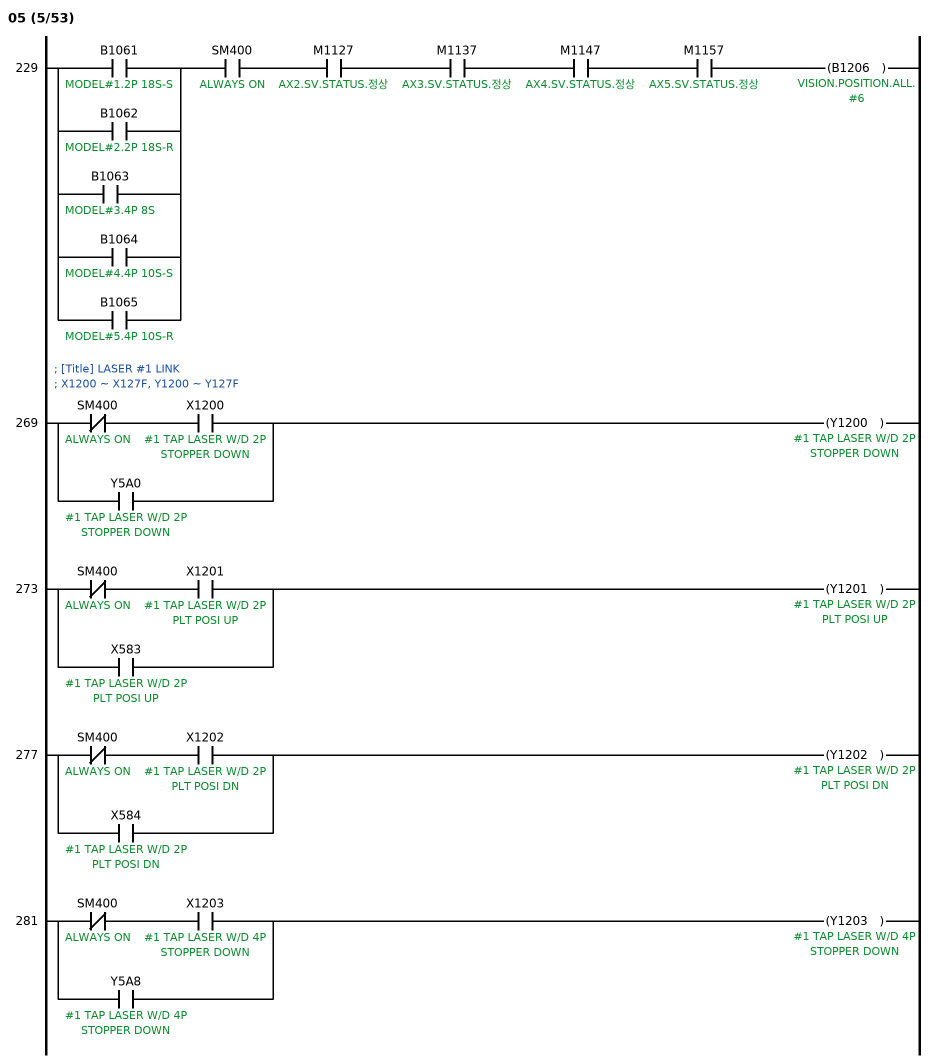
229   LD      B1061  ; MODEL#1.2P 18S-S
      OR      B1062  ; MODEL#2.2P 18S-R
      OR      B1063  ; MODEL#3.4P 8S
      OR      B1064  ; MODEL#4.4P 10S-S
      OR      B1065  ; MODEL#5.4P 10S-R
      AND     SM400  ; ALWAYS ON
      AND     M1127  ; AX2.SV.STATUS.정상
      AND     M1137  ; AX3.SV.STATUS.정상
      AND     M1147  ; AX4.SV.STATUS.정상
      AND     M1157  ; AX5.SV.STATUS.정상
      OUT     B1206  ; VISION.POSITION.ALL.#6
; [Title] LASER #1 LINK
; X1200 ~ X127F, Y1200 ~ Y127F
269   LDI     SM400  ; ALWAYS ON
      AND     X1200  ; #1 TAP LASER W/D 2P STOPPER DOWN
      OR      Y5A0  ; #1 TAP LASER W/D 2P STOPPER DOWN
      OUT     Y1200  ; #1 TAP LASER W/D 2P STOPPER DOWN
273   LDI     SM400  ; ALWAYS ON
      AND     X1201  ; #1 TAP LASER W/D 2P PLT POSI UP
      OR      X583  ; #1 TAP LASER W/D 2P PLT POSI UP
      OUT     Y1201  ; #1 TAP LASER W/D 2P PLT POSI UP
277   LDI     SM400  ; ALWAYS ON
      AND     X1202  ; #1 TAP LASER W/D 2P PLT POSI DN
      OR      X584  ; #1 TAP LASER W/D 2P PLT POSI DN
      OUT     Y1202  ; #1 TAP LASER W/D 2P PLT POSI DN
281   LDI     SM400  ; ALWAYS ON
      AND     X1203  ; #1 TAP LASER W/D 4P STOPPER DOWN
      OR      Y5A8  ; #1 TAP LASER W/D 4P STOPPER DOWN
      OUT     Y1203  ; #1 TAP LASER W/D 4P STOPPER DOWN
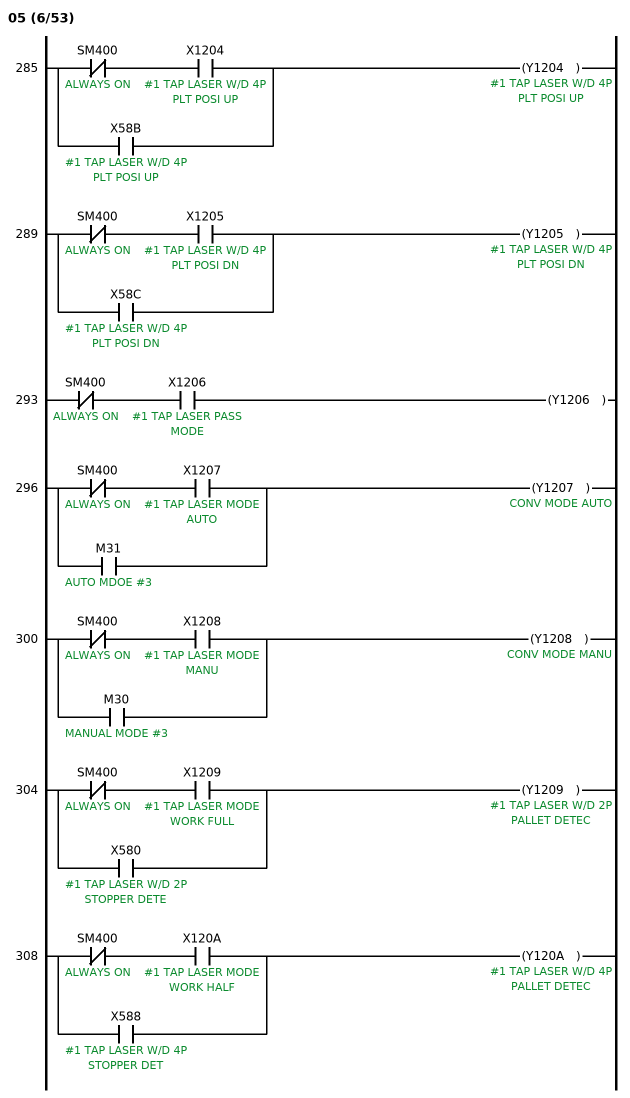
285   LDI     SM400  ; ALWAYS ON
      AND     X1204  ; #1 TAP LASER W/D 4P PLT POSI UP
      OR      X58B  ; #1 TAP LASER W/D 4P PLT POSI UP
      OUT     Y1204  ; #1 TAP LASER W/D 4P PLT POSI UP
289   LDI     SM400  ; ALWAYS ON
      AND     X1205  ; #1 TAP LASER W/D 4P PLT POSI DN
      OR      X58C  ; #1 TAP LASER W/D 4P PLT POSI DN
      OUT     Y1205  ; #1 TAP LASER W/D 4P PLT POSI DN
293   LDI     SM400  ; ALWAYS ON
      AND     X1206  ; #1 TAP LASER PASS MODE
      OUT     Y1206
296   LDI     SM400  ; ALWAYS ON
      AND     X1207  ; #1 TAP LASER MODE AUTO
      OR      M31  ; AUTO MDOE #3
      OUT     Y1207  ; CONV MODE AUTO
300   LDI     SM400  ; ALWAYS ON
      AND     X1208  ; #1 TAP LASER MODE MANU
      OR      M30  ; MANUAL MODE #3
      OUT     Y1208  ; CONV MODE MANU
304   LDI     SM400  ; ALWAYS ON
      AND     X1209  ; #1 TAP LASER MODE WORK FULL
      OR      X580  ; #1 TAP LASER W/D 2P STOPPER DETE
      OUT     Y1209  ; #1 TAP LASER W/D 2P PALLET DETEC
308   LDI     SM400  ; ALWAYS ON
      AND     X120A  ; #1 TAP LASER MODE WORK HALF
      OR      X588  ; #1 TAP LASER W/D 4P STOPPER DET
      OUT     Y120A  ; #1 TAP LASER W/D 4P PALLET DETEC
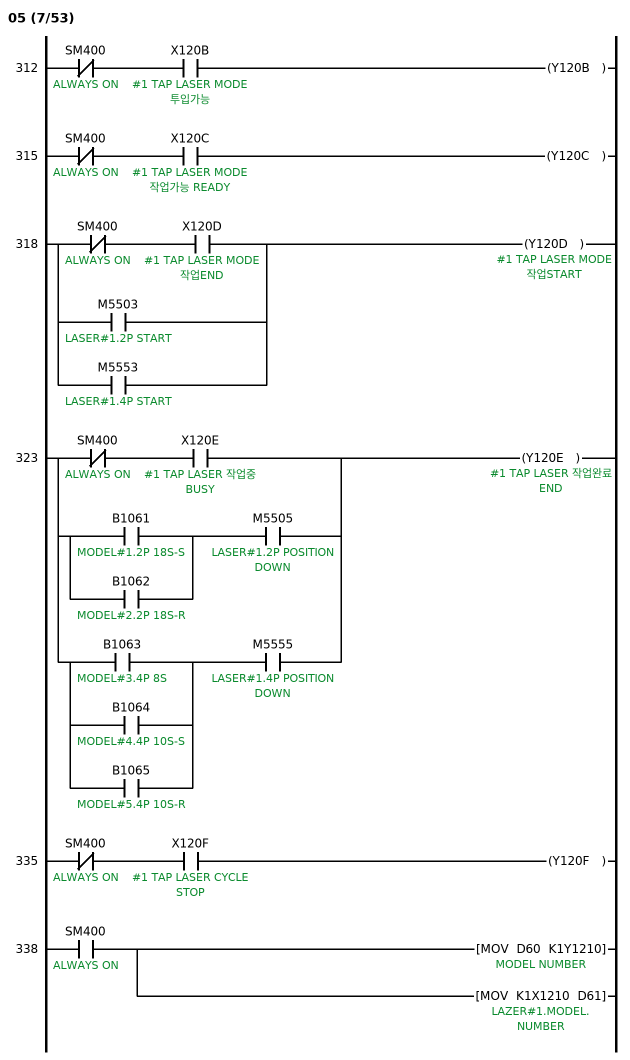
312   LDI     SM400  ; ALWAYS ON
      AND     X120B  ; #1 TAP LASER MODE 투입가능
      OUT     Y120B
315   LDI     SM400  ; ALWAYS ON
      AND     X120C  ; #1 TAP LASER MODE 작업가능 READY
      OUT     Y120C
318   LDI     SM400  ; ALWAYS ON
      AND     X120D  ; #1 TAP LASER MODE 작업END
      OR      M5503  ; LASER#1.2P START
      OR      M5553  ; LASER#1.4P START
      OUT     Y120D  ; #1 TAP LASER MODE 작업START
323   LDI     SM400  ; ALWAYS ON
      AND     X120E  ; #1 TAP LASER 작업중 BUSY
      LD      B1061  ; MODEL#1.2P 18S-S
      OR      B1062  ; MODEL#2.2P 18S-R
      AND     M5505  ; LASER#1.2P POSITION DOWN
      ORB
      LD      B1063  ; MODEL#3.4P 8S
      OR      B1064  ; MODEL#4.4P 10S-S
      OR      B1065  ; MODEL#5.4P 10S-R
      AND     M5555  ; LASER#1.4P POSITION DOWN
      ORB
      OUT     Y120E  ; #1 TAP LASER 작업완료 END
335   LDI     SM400  ; ALWAYS ON
      AND     X120F  ; #1 TAP LASER CYCLE STOP
      OUT     Y120F
338   LD      SM400  ; ALWAYS ON
      MOV     D60 K1Y1210
      MOV     K1X1210 D61  ; LAZER#1.MODEL.NUMBER
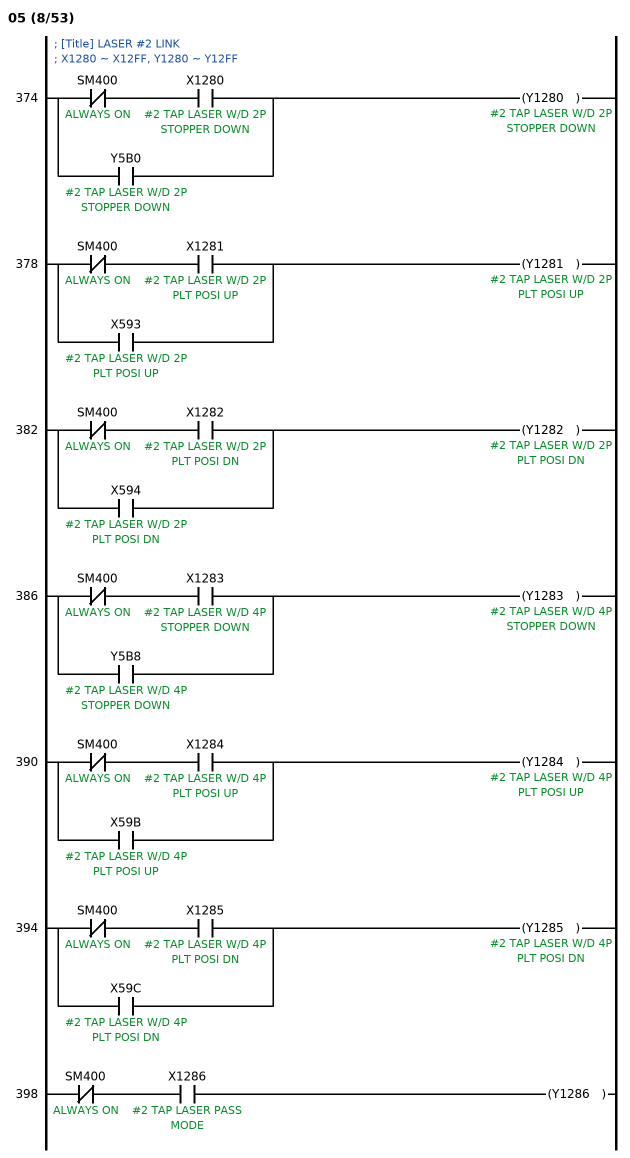
; [Title] LASER #2 LINK
; X1280 ~ X12FF, Y1280 ~ Y12FF
374   LDI     SM400  ; ALWAYS ON
      AND     X1280  ; #2 TAP LASER W/D 2P STOPPER DOWN
      OR      Y5B0  ; #2 TAP LASER W/D 2P STOPPER DOWN
      OUT     Y1280  ; #2 TAP LASER W/D 2P STOPPER DOWN
378   LDI     SM400  ; ALWAYS ON
      AND     X1281  ; #2 TAP LASER W/D 2P PLT POSI UP
      OR      X593  ; #2 TAP LASER W/D 2P PLT POSI UP
      OUT     Y1281  ; #2 TAP LASER W/D 2P PLT POSI UP
382   LDI     SM400  ; ALWAYS ON
      AND     X1282  ; #2 TAP LASER W/D 2P PLT POSI DN
      OR      X594  ; #2 TAP LASER W/D 2P PLT POSI DN
      OUT     Y1282  ; #2 TAP LASER W/D 2P PLT POSI DN
386   LDI     SM400  ; ALWAYS ON
      AND     X1283  ; #2 TAP LASER W/D 4P STOPPER DOWN
      OR      Y5B8  ; #2 TAP LASER W/D 4P STOPPER DOWN
      OUT     Y1283  ; #2 TAP LASER W/D 4P STOPPER DOWN
390   LDI     SM400  ; ALWAYS ON
      AND     X1284  ; #2 TAP LASER W/D 4P PLT POSI UP
      OR      X59B  ; #2 TAP LASER W/D 4P PLT POSI UP
      OUT     Y1284  ; #2 TAP LASER W/D 4P PLT POSI UP
394   LDI     SM400  ; ALWAYS ON
      AND     X1285  ; #2 TAP LASER W/D 4P PLT POSI DN
      OR      X59C  ; #2 TAP LASER W/D 4P PLT POSI DN
      OUT     Y1285  ; #2 TAP LASER W/D 4P PLT POSI DN
398   LDI     SM400  ; ALWAYS ON
      AND     X1286  ; #2 TAP LASER PASS MODE
      OUT     Y1286
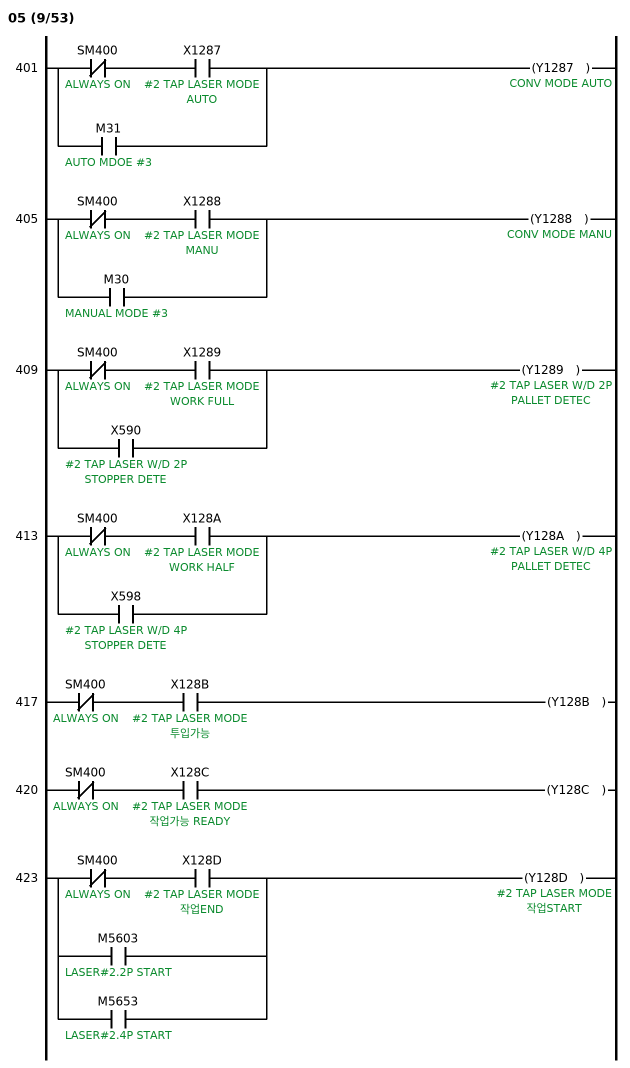
401   LDI     SM400  ; ALWAYS ON
      AND     X1287  ; #2 TAP LASER MODE AUTO
      OR      M31  ; AUTO MDOE #3
      OUT     Y1287  ; CONV MODE AUTO
405   LDI     SM400  ; ALWAYS ON
      AND     X1288  ; #2 TAP LASER MODE MANU
      OR      M30  ; MANUAL MODE #3
      OUT     Y1288  ; CONV MODE MANU
409   LDI     SM400  ; ALWAYS ON
      AND     X1289  ; #2 TAP LASER MODE WORK FULL
      OR      X590  ; #2 TAP LASER W/D 2P STOPPER DETE
      OUT     Y1289  ; #2 TAP LASER W/D 2P PALLET DETEC
413   LDI     SM400  ; ALWAYS ON
      AND     X128A  ; #2 TAP LASER MODE WORK HALF
      OR      X598  ; #2 TAP LASER W/D 4P STOPPER DETE
      OUT     Y128A  ; #2 TAP LASER W/D 4P PALLET DETEC
417   LDI     SM400  ; ALWAYS ON
      AND     X128B  ; #2 TAP LASER MODE 투입가능
      OUT     Y128B
420   LDI     SM400  ; ALWAYS ON
      AND     X128C  ; #2 TAP LASER MODE 작업가능 READY
      OUT     Y128C
423   LDI     SM400  ; ALWAYS ON
      AND     X128D  ; #2 TAP LASER MODE 작업END
      OR      M5603  ; LASER#2.2P START
      OR      M5653  ; LASER#2.4P START
      OUT     Y128D  ; #2 TAP LASER MODE 작업START
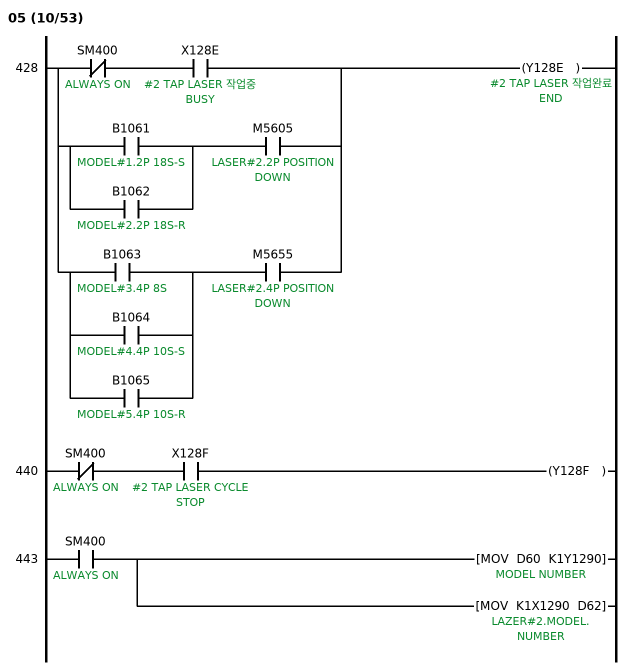
428   LDI     SM400  ; ALWAYS ON
      AND     X128E  ; #2 TAP LASER 작업중 BUSY
      LD      B1061  ; MODEL#1.2P 18S-S
      OR      B1062  ; MODEL#2.2P 18S-R
      AND     M5605  ; LASER#2.2P POSITION DOWN
      ORB
      LD      B1063  ; MODEL#3.4P 8S
      OR      B1064  ; MODEL#4.4P 10S-S
      OR      B1065  ; MODEL#5.4P 10S-R
      AND     M5655  ; LASER#2.4P POSITION DOWN
      ORB
      OUT     Y128E  ; #2 TAP LASER 작업완료 END
440   LDI     SM400  ; ALWAYS ON
      AND     X128F  ; #2 TAP LASER CYCLE STOP
      OUT     Y128F
443   LD      SM400  ; ALWAYS ON
      MOV     D60 K1Y1290
      MOV     K1X1290 D62  ; LAZER#2.MODEL.NUMBER
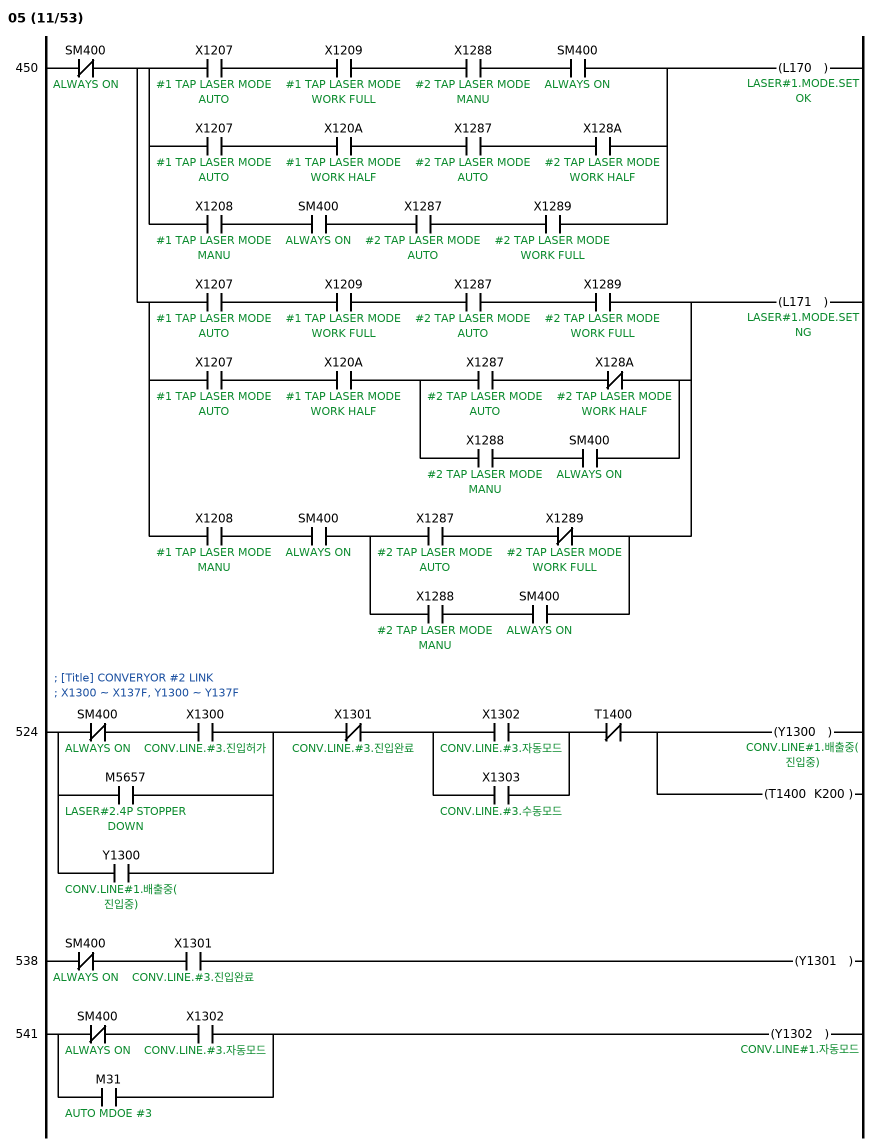
450   LDI     SM400  ; ALWAYS ON
      MPS
      LD      X1207  ; #1 TAP LASER MODE AUTO
      AND     X1209  ; #1 TAP LASER MODE WORK FULL
      AND     X1288  ; #2 TAP LASER MODE MANU
      AND     SM400  ; ALWAYS ON
      LD      X1207  ; #1 TAP LASER MODE AUTO
      AND     X120A  ; #1 TAP LASER MODE WORK HALF
      AND     X1287  ; #2 TAP LASER MODE AUTO
      AND     X128A  ; #2 TAP LASER MODE WORK HALF
      ORB
      LD      X1208  ; #1 TAP LASER MODE MANU
      AND     SM400  ; ALWAYS ON
      AND     X1287  ; #2 TAP LASER MODE AUTO
      AND     X1289  ; #2 TAP LASER MODE WORK FULL
      ORB
      ANB
      OUT     L170  ; LASER#1.MODE.SET OK
      MPP
      LD      X1207  ; #1 TAP LASER MODE AUTO
      AND     X1209  ; #1 TAP LASER MODE WORK FULL
      AND     X1287  ; #2 TAP LASER MODE AUTO
      AND     X1289  ; #2 TAP LASER MODE WORK FULL
      LD      X1207  ; #1 TAP LASER MODE AUTO
      AND     X120A  ; #1 TAP LASER MODE WORK HALF
      LD      X1287  ; #2 TAP LASER MODE AUTO
      ANI     X128A  ; #2 TAP LASER MODE WORK HALF
      LD      X1288  ; #2 TAP LASER MODE MANU
      AND     SM400  ; ALWAYS ON
      ORB
      ANB
      ORB
      LD      X1208  ; #1 TAP LASER MODE MANU
      AND     SM400  ; ALWAYS ON
      LD      X1287  ; #2 TAP LASER MODE AUTO
      ANI     X1289  ; #2 TAP LASER MODE WORK FULL
      LD      X1288  ; #2 TAP LASER MODE MANU
      AND     SM400  ; ALWAYS ON
      ORB
      ANB
      ORB
      ANB
      OUT     L171  ; LASER#1.MODE.SET NG
; [Title] CONVERYOR #2 LINK
; X1300 ~ X137F, Y1300 ~ Y137F
524   LDI     SM400  ; ALWAYS ON
      AND     X1300  ; CONV.LINE.#3.진입허가
      OR      M5657  ; LASER#2.4P STOPPER DOWN
      OR      Y1300  ; CONV.LINE#1.배출중(진입중)
      ANI     X1301  ; CONV.LINE.#3.진입완료
      LD      X1302  ; CONV.LINE.#3.자동모드
      OR      X1303  ; CONV.LINE.#3.수동모드
      ANB
      ANI     T1400
      OUT     Y1300  ; CONV.LINE#1.배출중(진입중)
      OUT     T1400 K200
538   LDI     SM400  ; ALWAYS ON
      AND     X1301  ; CONV.LINE.#3.진입완료
      OUT     Y1301
541   LDI     SM400  ; ALWAYS ON
      AND     X1302  ; CONV.LINE.#3.자동모드
      OR      M31  ; AUTO MDOE #3
      OUT     Y1302  ; CONV.LINE#1.자동모드
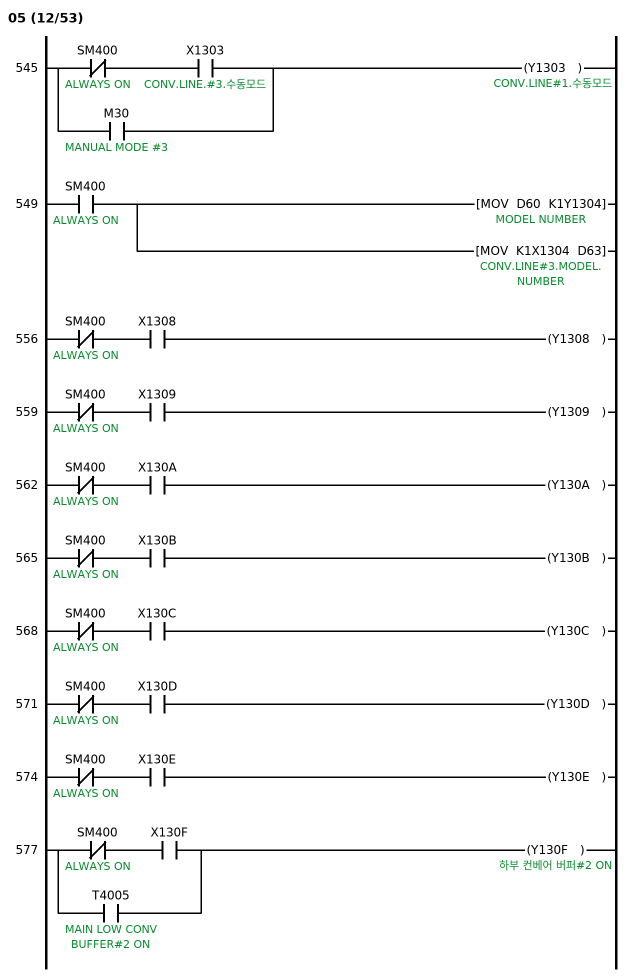
545   LDI     SM400  ; ALWAYS ON
      AND     X1303  ; CONV.LINE.#3.수동모드
      OR      M30  ; MANUAL MODE #3
      OUT     Y1303  ; CONV.LINE#1.수동모드
549   LD      SM400  ; ALWAYS ON
      MOV     D60 K1Y1304  ; MODEL BIT #1
      MOV     K1X1304 D63  ; MODEL BIT #1 / CONV.LINE#3.MODEL.NUMBER
556   LDI     SM400  ; ALWAYS ON
      AND     X1308
      OUT     Y1308
559   LDI     SM400  ; ALWAYS ON
      AND     X1309
      OUT     Y1309
562   LDI     SM400  ; ALWAYS ON
      AND     X130A
      OUT     Y130A
565   LDI     SM400  ; ALWAYS ON
      AND     X130B
      OUT     Y130B
568   LDI     SM400  ; ALWAYS ON
      AND     X130C
      OUT     Y130C
571   LDI     SM400  ; ALWAYS ON
      AND     X130D
      OUT     Y130D
574   LDI     SM400  ; ALWAYS ON
      AND     X130E
      OUT     Y130E
577   LDI     SM400  ; ALWAYS ON
      AND     X130F
      OR      T4005  ; MAIN LOW CONV BUFFER#2 ON
      OUT     Y130F  ; 하부 컨베어 버퍼#2 ON
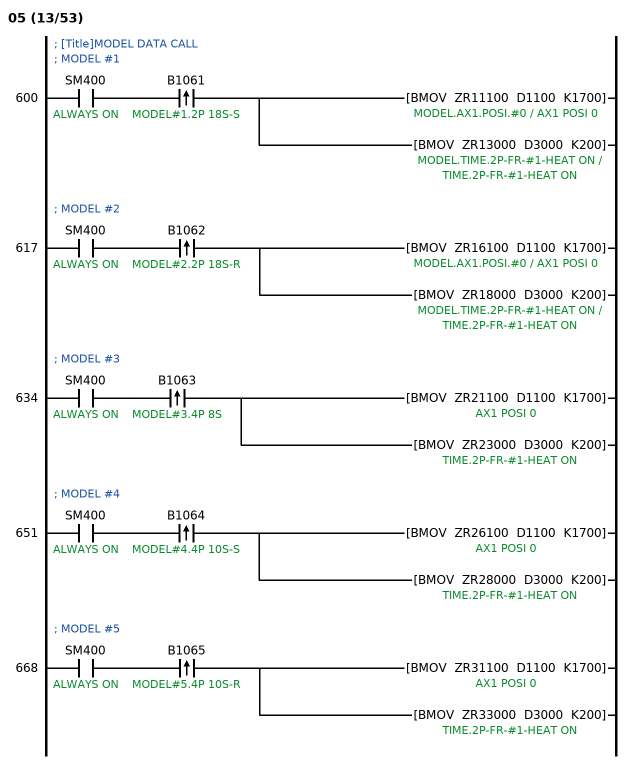
; [Title]MODEL DATA CALL
; MODEL #1
600   LD      SM400  ; ALWAYS ON
      ANDP    B1061  ; MODEL#1.2P 18S-S
      BMOV    ZR11100 D1100 K1700  ; MODEL.AX1.POSI.#0 / AX1 POSI 0
      BMOV    ZR13000 D3000 K200  ; MODEL.TIME.2P-FR-#1-HEAT ON / TIME.2P-FR-#1-HEAT ON
; MODEL #2
617   LD      SM400  ; ALWAYS ON
      ANDP    B1062  ; MODEL#2.2P 18S-R
      BMOV    ZR16100 D1100 K1700  ; MODEL.AX1.POSI.#0
      BMOV    ZR18000 D3000 K200  ; MODEL.TIME.2P-FR-#1-HEAT ON
; MODEL #3
634   LD      SM400  ; ALWAYS ON
      ANDP    B1063  ; MODEL#3.4P 8S
      BMOV    ZR21100 D1100 K1700
      BMOV    ZR23000 D3000 K200
; MODEL #4
651   LD      SM400  ; ALWAYS ON
      ANDP    B1064  ; MODEL#4.4P 10S-S
      BMOV    ZR26100 D1100 K1700
      BMOV    ZR28000 D3000 K200
; MODEL #5
668   LD      SM400  ; ALWAYS ON
      ANDP    B1065  ; MODEL#5.4P 10S-R
      BMOV    ZR31100 D1100 K1700
      BMOV    ZR33000 D3000 K200
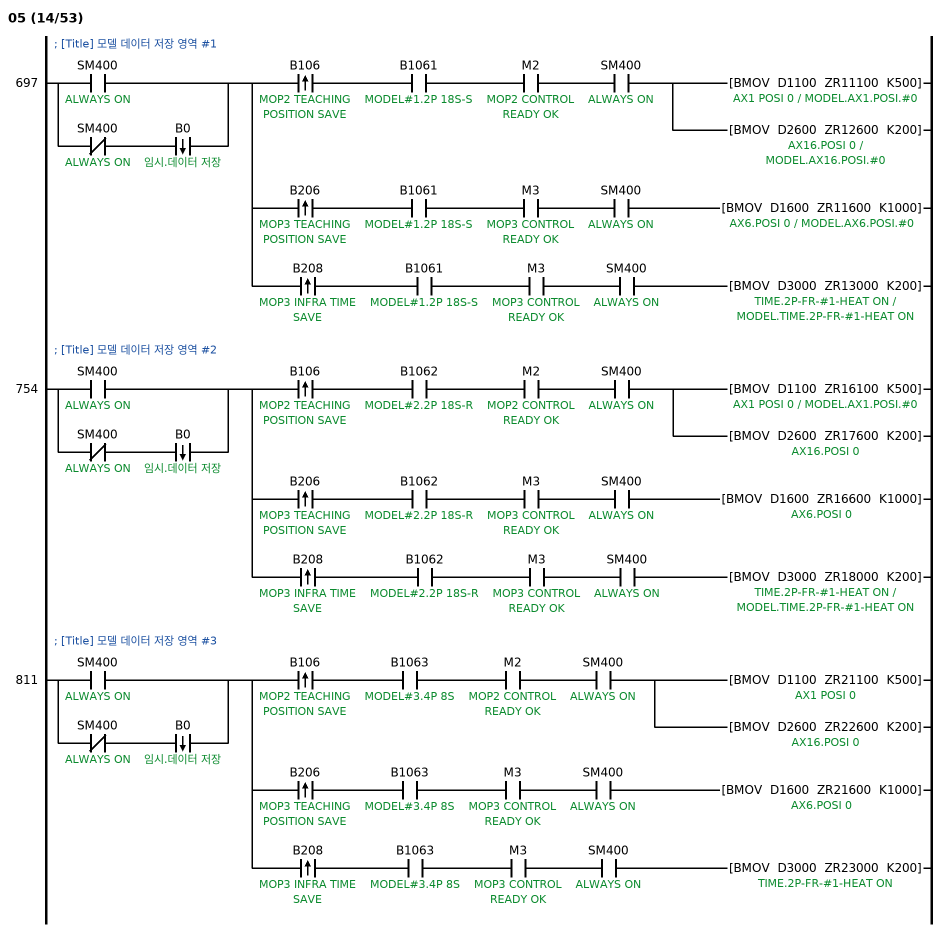
; [Title] 모델 데이터 저장 영역 #1
697   LD      SM400  ; ALWAYS ON
      LDI     SM400  ; ALWAYS ON
      ANDF    B0  ; 임시.데이터 저장
      ORB
      MPS
      ANDP    B106  ; MOP2 TEACHING POSITION SAVE
      AND     B1061  ; MODEL#1.2P 18S-S
      AND     M2  ; MOP2 CONTROL READY OK
      AND     SM400  ; ALWAYS ON
      BMOV    D1100 ZR11100 K500
      BMOV    D2600 ZR12600 K200  ; AX16.POSI 0 / MODEL.AX16.POSI.#0
      MRD
      ANDP    B206  ; MOP3 TEACHING POSITION SAVE
      AND     B1061  ; MODEL#1.2P 18S-S
      AND     M3  ; MOP3 CONTROL READY OK
      AND     SM400  ; ALWAYS ON
      BMOV    D1600 ZR11600 K1000  ; AX6.POSI 0 / MODEL.AX6.POSI.#0
      MPP
      ANDP    B208  ; MOP3 INFRA TIME SAVE
      AND     B1061  ; MODEL#1.2P 18S-S
      AND     M3  ; MOP3 CONTROL READY OK
      AND     SM400  ; ALWAYS ON
      BMOV    D3000 ZR13000 K200
; [Title] 모델 데이터 저장 영역 #2
754   LD      SM400  ; ALWAYS ON
      LDI     SM400  ; ALWAYS ON
      ANDF    B0  ; 임시.데이터 저장
      ORB
      MPS
      ANDP    B106  ; MOP2 TEACHING POSITION SAVE
      AND     B1062  ; MODEL#2.2P 18S-R
      AND     M2  ; MOP2 CONTROL READY OK
      AND     SM400  ; ALWAYS ON
      BMOV    D1100 ZR16100 K500
      BMOV    D2600 ZR17600 K200
      MRD
      ANDP    B206  ; MOP3 TEACHING POSITION SAVE
      AND     B1062  ; MODEL#2.2P 18S-R
      AND     M3  ; MOP3 CONTROL READY OK
      AND     SM400  ; ALWAYS ON
      BMOV    D1600 ZR16600 K1000
      MPP
      ANDP    B208  ; MOP3 INFRA TIME SAVE
      AND     B1062  ; MODEL#2.2P 18S-R
      AND     M3  ; MOP3 CONTROL READY OK
      AND     SM400  ; ALWAYS ON
      BMOV    D3000 ZR18000 K200
; [Title] 모델 데이터 저장 영역 #3
811   LD      SM400  ; ALWAYS ON
      LDI     SM400  ; ALWAYS ON
      ANDF    B0  ; 임시.데이터 저장
      ORB
      MPS
      ANDP    B106  ; MOP2 TEACHING POSITION SAVE
      AND     B1063  ; MODEL#3.4P 8S
      AND     M2  ; MOP2 CONTROL READY OK
      AND     SM400  ; ALWAYS ON
      BMOV    D1100 ZR21100 K500
      BMOV    D2600 ZR22600 K200
      MRD
      ANDP    B206  ; MOP3 TEACHING POSITION SAVE
      AND     B1063  ; MODEL#3.4P 8S
      AND     M3  ; MOP3 CONTROL READY OK
      AND     SM400  ; ALWAYS ON
      BMOV    D1600 ZR21600 K1000
      MPP
      ANDP    B208  ; MOP3 INFRA TIME SAVE
      AND     B1063  ; MODEL#3.4P 8S
      AND     M3  ; MOP3 CONTROL READY OK
      AND     SM400  ; ALWAYS ON
      BMOV    D3000 ZR23000 K200
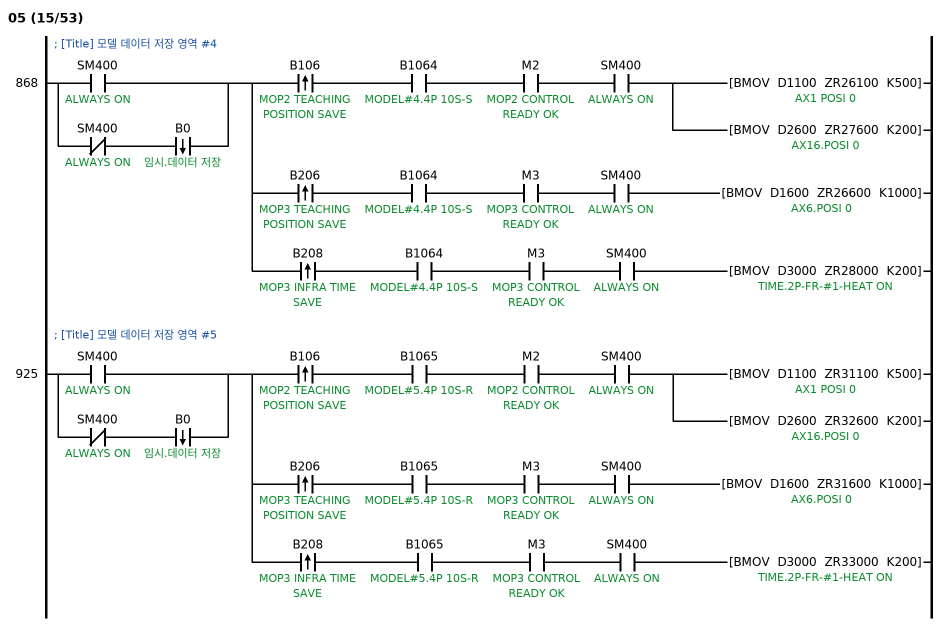
; [Title] 모델 데이터 저장 영역 #4
868   LD      SM400  ; ALWAYS ON
      LDI     SM400  ; ALWAYS ON
      ANDF    B0  ; 임시.데이터 저장
      ORB
      MPS
      ANDP    B106  ; MOP2 TEACHING POSITION SAVE
      AND     B1064  ; MODEL#4.4P 10S-S
      AND     M2  ; MOP2 CONTROL READY OK
      AND     SM400  ; ALWAYS ON
      BMOV    D1100 ZR26100 K500
      BMOV    D2600 ZR27600 K200
      MRD
      ANDP    B206  ; MOP3 TEACHING POSITION SAVE
      AND     B1064  ; MODEL#4.4P 10S-S
      AND     M3  ; MOP3 CONTROL READY OK
      AND     SM400  ; ALWAYS ON
      BMOV    D1600 ZR26600 K1000
      MPP
      ANDP    B208  ; MOP3 INFRA TIME SAVE
      AND     B1064  ; MODEL#4.4P 10S-S
      AND     M3  ; MOP3 CONTROL READY OK
      AND     SM400  ; ALWAYS ON
      BMOV    D3000 ZR28000 K200
; [Title] 모델 데이터 저장 영역 #5
925   LD      SM400  ; ALWAYS ON
      LDI     SM400  ; ALWAYS ON
      ANDF    B0  ; 임시.데이터 저장
      ORB
      MPS
      ANDP    B106  ; MOP2 TEACHING POSITION SAVE
      AND     B1065  ; MODEL#5.4P 10S-R
      AND     M2  ; MOP2 CONTROL READY OK
      AND     SM400  ; ALWAYS ON
      BMOV    D1100 ZR31100 K500
      BMOV    D2600 ZR32600 K200
      MRD
      ANDP    B206  ; MOP3 TEACHING POSITION SAVE
      AND     B1065  ; MODEL#5.4P 10S-R
      AND     M3  ; MOP3 CONTROL READY OK
      AND     SM400  ; ALWAYS ON
      BMOV    D1600 ZR31600 K1000
      MPP
      ANDP    B208  ; MOP3 INFRA TIME SAVE
      AND     B1065  ; MODEL#5.4P 10S-R
      AND     M3  ; MOP3 CONTROL READY OK
      AND     SM400  ; ALWAYS ON
      BMOV    D3000 ZR33000 K200
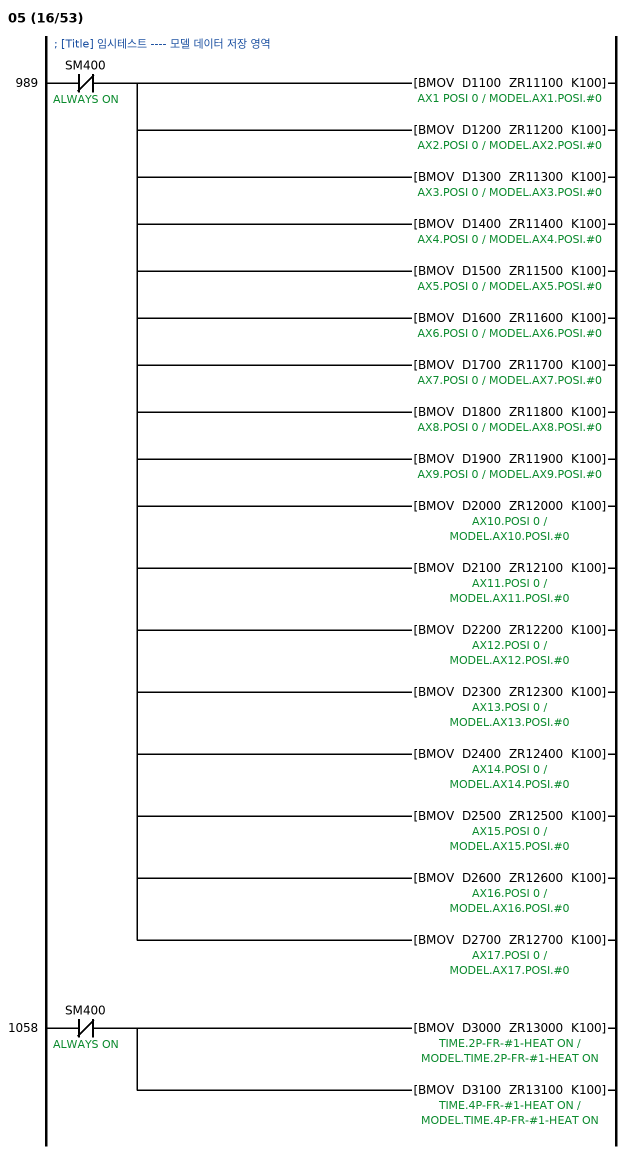
; [Title] 임시테스트 ---- 모델 데이터 저장 영역
989   LDI     SM400  ; ALWAYS ON
      BMOV    D1100 ZR11100 K100
      BMOV    D1200 ZR11200 K100  ; AX2.POSI 0 / MODEL.AX2.POSI.#0
      BMOV    D1300 ZR11300 K100  ; AX3.POSI 0 / MODEL.AX3.POSI.#0
      BMOV    D1400 ZR11400 K100  ; AX4.POSI 0 / MODEL.AX4.POSI.#0
      BMOV    D1500 ZR11500 K100  ; AX5.POSI 0 / MODEL.AX5.POSI.#0
      BMOV    D1600 ZR11600 K100
      BMOV    D1700 ZR11700 K100  ; AX7.POSI 0 / MODEL.AX7.POSI.#0
      BMOV    D1800 ZR11800 K100  ; AX8.POSI 0 / MODEL.AX8.POSI.#0
      BMOV    D1900 ZR11900 K100  ; AX9.POSI 0 / MODEL.AX9.POSI.#0
      BMOV    D2000 ZR12000 K100  ; AX10.POSI 0 / MODEL.AX10.POSI.#0
      BMOV    D2100 ZR12100 K100  ; AX11.POSI 0 / MODEL.AX11.POSI.#0
      BMOV    D2200 ZR12200 K100  ; AX12.POSI 0 / MODEL.AX12.POSI.#0
      BMOV    D2300 ZR12300 K100  ; AX13.POSI 0 / MODEL.AX13.POSI.#0
      BMOV    D2400 ZR12400 K100  ; AX14.POSI 0 / MODEL.AX14.POSI.#0
      BMOV    D2500 ZR12500 K100  ; AX15.POSI 0 / MODEL.AX15.POSI.#0
      BMOV    D2600 ZR12600 K100
      BMOV    D2700 ZR12700 K100  ; AX17.POSI 0 / MODEL.AX17.POSI.#0
1058  LDI     SM400  ; ALWAYS ON
      BMOV    D3000 ZR13000 K100
      BMOV    D3100 ZR13100 K100  ; TIME.4P-FR-#1-HEAT ON / MODEL.TIME.4P-FR-#1-HEAT ON
